LIN {X 0,Y 317.653,Z 381.301,A -85,B 0,C 180,E1 -15906.448,E2 -15906.448} C_VEL
LIN {X 0,Y 316.259,Z 393.2,A -85,B 0,C 180,E1 -15907.203,E2 -15907.203} C_VEL
LIN {X 0,Y 314.587,Z 404.894,A -85,B 0,C 180,E1 -15908.2,E2 -15908.2} C_VEL
LIN {X 0,Y 312.768,Z 416.27,A -85,B 0,C 180,E1 -15909.448,E2 -15909.448} C_VEL
LIN {X 0,Y 310.949,Z 426.626,A -85,B 0,C 180,E1 -15910.871,E2 -15910.871} C_VEL
LIN {X 0,Y 309.178,Z 435.992,A -85,B 0,C 180,E1 -15912.473,E2 -15912.473} C_VEL
LIN {X 0,Y 307.511,Z 445.132,A -85,B 0,C 180,E1 -15914.424,E2 -15914.424} C_VEL
LIN {X 0,Y 306.132,Z 452.545,A -85,B 0,C 180,E1 -15916.391,E2 -15916.391} C_VEL
LIN {X 0,Y 305.102,Z 457.603,A -85,B 0,C 180,E1 -15918.036,E2 -15918.036} C_VEL
LIN {X 0,Y 304.379,Z 462.545,A -85,B 0,C 180,E1 -15920.029,E2 -15920.029} C_VEL
LIN {X 0,Y 303.921,Z 466.357,A -85,B 0,C 180,E1 -15922.025,E2 -15922.025} C_VEL
LIN {X 0,Y 303.627,Z 469.641,A -85,B 0,C 180,E1 -15924.456,E2 -15924.456} C_VEL
LIN {X 0,Y 303.64,Z 470.96,A -85,B 0,C 180,E1 -15926.019,E2 -15926.019} C_VEL
LIN {X 0,Y 303.653,Z 471.66,A -85,B 0,C 180,E1 -15927.347,E2 -15927.347} C_VEL
LIN {X 0,Y 303.684,Z 471.954,A -85,B 0,C 180,E1 -15928.674,E2 -15928.674} C_VEL
LIN {X 0,Y 303.768,Z 471.795,A -85,B 0,C 180,E1 -15930,E2 -15930} C_VEL
LIN {X 0,Y 303.712,Z 471.218,A -85,B 0,C 180,E1 -15931.326,E2 -15931.326} C_VEL
LIN {X 0,Y 303.68,Z 470.233,A -85,B 0,C 180,E1 -15932.652,E2 -15932.652} C_VEL
LIN {X 0,Y 303.699,Z 468.813,A -85,B 0,C 180,E1 -15933.98,E2 -15933.98} C_VEL
LIN {X 0,Y 303.735,Z 466.181,A -85,B 0,C 180,E1 -15935.751,E2 -15935.751} C_VEL
LIN {X 0,Y 303.933,Z 461.681,A -85,B 0,C 180,E1 -15937.974,E2 -15937.974} C_VEL
LIN {X 0,Y 304.394,Z 455.299,A -85,B 0,C 180,E1 -15940.307,E2 -15940.307} C_VEL
LIN {X 0,Y 305.068,Z 448.32,A -85,B 0,C 180,E1 -15942.302,E2 -15942.302} C_VEL
LIN {X 0,Y 305.863,Z 441.179,A -85,B 0,C 180,E1 -15943.959,E2 -15943.959} C_VEL
LIN {X 0,Y 306.821,Z 433.215,A -85,B 0,C 180,E1 -15945.491,E2 -15945.491} C_VEL
LIN {X 0,Y 307.985,Z 423.186,A -85,B 0,C 180,E1 -15947.066,E2 -15947.066} C_VEL
LIN {X 0,Y 309.15,Z 412.766,A -85,B 0,C 180,E1 -15948.384,E2 -15948.384} C_VEL
LIN {X 0,Y 310.352,Z 401.577,A -85,B 0,C 180,E1 -15949.51,E2 -15949.51} C_VEL
LIN {X 0,Y 311.498,Z 389.171,A -85,B 0,C 180,E1 -15950.467,E2 -15950.467} C_VEL
LIN {X 0,Y 312.472,Z 375.35,A -85,B 0,C 180,E1 -15951.219,E2 -15951.219} C_VEL
LIN {X 0,Y 313.086,Z 362.94,A -85,B 0,C 180,E1 -15951.65,E2 -15951.65} C_VEL
LIN {X 0,Y 314.499,Z 301.548,A -85,B 0,C 180,E1 -15953.24,E2 -15953.24} C_VEL
LIN {X 0,Y 309.032,Z 259.907,A -85,B 0,C 180,E1 -15954.774,E2 -15954.774} C_VEL
LIN {X 0,Y 309.789,Z 252.83,A -85,B 0,C 180,E1 -15956.616,E2 -15956.616} C_VEL
LIN {X 0,Y 308.031,Z 243.339,A -85,B 0,C 180,E1 -15959.295,E2 -15959.295} C_VEL
LIN {X 0,Y 305.483,Z 231.433,A -85,B 0,C 180,E1 -15962.821,E2 -15962.821} C_VEL
LIN {X 0,Y 305.445,Z 231.435,A -85,B 0,C 180,E1 -15966.739,E2 -15966.739} C_VEL
LIN {X 0,Y 305.44,Z 231.436,A -85,B 0,C 180,E1 -15970.596,E2 -15970.596} C_VEL
LIN {X 0,Y 305.408,Z 231.444,A -85,B 0,C 180,E1 -15973.652,E2 -15973.652} C_VEL
LIN {X 0,Y 305.435,Z 231.439,A -85,B 0,C 180,E1 -15977.411,E2 -15977.411} C_VEL
LIN {X 0,Y 305.453,Z 231.438,A -85,B 0,C 180,E1 -15981.594,E2 -15981.594} C_VEL
LIN {X 0,Y 305.437,Z 231.436,A -85,B 0,C 180,E1 -15984.883,E2 -15984.883} C_VEL
LIN {X 0,Y 305.415,Z 231.439,A -85,B 0,C 180,E1 -15988.356,E2 -15988.356} C_VEL
LIN {X 0,Y 305.471,Z 231.434,A -85,B 0,C 180,E1 -15991.108,E2 -15991.108} C_VEL
LIN {X 0,Y 305.524,Z 231.424,A -85,B 0,C 180,E1 -15994.083,E2 -15994.083} C_VEL
LIN {X 0,Y 305.43,Z 231.437,A -85,B 0,C 180,E1 -15998.397,E2 -15998.397} C_VEL
LIN {X 0,Y 305.483,Z 231.434,A -85,B 0,C 180,E1 -16001.21,E2 -16001.21} C_VEL
LIN {X 0,Y 305.591,Z 231.419,A -85,B 0,C 180,E1 -16005.346,E2 -16005.346} C_VEL
LIN {X 0,Y 305.599,Z 231.418,A -85,B 0,C 180,E1 -16009.398,E2 -16009.398} C_VEL
LIN {X 0,Y 305.749,Z 231.397,A -85,B 0,C 180,E1 -16012.072,E2 -16012.072} C_VEL
LIN {X 0,Y 305.641,Z 231.412,A -85,B 0,C 180,E1 -16014.722,E2 -16014.722} C_VEL
LIN {X 0,Y 305.915,Z 231.376,A -85,B 0,C 180,E1 -16018.683,E2 -16018.683} C_VEL
LIN {X 0,Y 305.917,Z 231.376,A -85,B 0,C 180,E1 -16021.316,E2 -16021.316} C_VEL
LIN {X 0,Y 305.805,Z 231.393,A -85,B 0,C 180,E1 -16026.598,E2 -16026.598} C_VEL
LIN {X 0,Y 305.664,Z 231.408,A -85,B 0,C 180,E1 -16029.261,E2 -16029.261} C_VEL
LIN {X 0,Y 305.551,Z 231.421,A -85,B 0,C 180,E1 -16033.297,E2 -16033.297} C_VEL
LIN {X 0,Y 305.524,Z 231.423,A -85,B 0,C 180,E1 -16036.023,E2 -16036.023} C_VEL
LIN {X 0,Y 305.572,Z 231.414,A -85,B 0,C 180,E1 -16039.46,E2 -16039.46} C_VEL
LIN {X 0,Y 305.526,Z 231.424,A -85,B 0,C 180,E1 -16043.072,E2 -16043.072} C_VEL
LIN {X 0,Y 305.518,Z 231.428,A -85,B 0,C 180,E1 -16046.229,E2 -16046.229} C_VEL
LIN {X 0,Y 305.465,Z 231.433,A -85,B 0,C 180,E1 -16049.051,E2 -16049.051} C_VEL
LIN {X 0,Y 305.438,Z 231.435,A -85,B 0,C 180,E1 -16053.52,E2 -16053.52} C_VEL
LIN {X 0,Y 305.455,Z 231.431,A -85,B 0,C 180,E1 -16056.742,E2 -16056.742} C_VEL
LIN {X 0,Y 305.461,Z 231.43,A -85,B 0,C 180,E1 -16060.609,E2 -16060.609} C_VEL
LIN {X 0,Y 305.466,Z 231.432,A -85,B 0,C 180,E1 -16063.647,E2 -16063.647} C_VEL
LIN {X 0,Y 305.443,Z 231.435,A -85,B 0,C 180,E1 -16067.416,E2 -16067.416} C_VEL
LIN {X 0,Y 305.48,Z 231.432,A -85,B 0,C 180,E1 -16071.603,E2 -16071.603} C_VEL
LIN {X 0,Y 305.447,Z 231.433,A -85,B 0,C 180,E1 -16074.889,E2 -16074.889} C_VEL
LIN {X 0,Y 305.439,Z 231.434,A -85,B 0,C 180,E1 -16078.358,E2 -16078.358} C_VEL
LIN {X 0,Y 305.518,Z 231.425,A -85,B 0,C 180,E1 -16081.117,E2 -16081.117} C_VEL
LIN {X 0,Y 305.562,Z 231.422,A -85,B 0,C 180,E1 -16084.09,E2 -16084.09} C_VEL
LIN {X 0,Y 305.494,Z 231.428,A -85,B 0,C 180,E1 -16088.405,E2 -16088.405} C_VEL
LIN {X 0,Y 305.585,Z 231.418,A -85,B 0,C 180,E1 -16091.22,E2 -16091.22} C_VEL
LIN {X 0,Y 305.645,Z 231.414,A -85,B 0,C 180,E1 -16095.351,E2 -16095.351} C_VEL
LIN {X 0,Y 305.635,Z 231.415,A -85,B 0,C 180,E1 -16099.401,E2 -16099.401} C_VEL
LIN {X 0,Y 305.806,Z 231.39,A -85,B 0,C 180,E1 -16102.075,E2 -16102.075} C_VEL
LIN {X 0,Y 305.685,Z 231.406,A -85,B 0,C 180,E1 -16104.724,E2 -16104.724} C_VEL
LIN {X 0,Y 305.956,Z 231.372,A -85,B 0,C 180,E1 -16108.684,E2 -16108.684} C_VEL
LIN {X 0,Y 305.954,Z 231.375,A -85,B 0,C 180,E1 -16111.316,E2 -16111.316} C_VEL
LIN {X 0,Y 305.684,Z 231.409,A -85,B 0,C 180,E1 -16115.276,E2 -16115.276} C_VEL
LIN {X 0,Y 305.799,Z 231.391,A -85,B 0,C 180,E1 -16117.925,E2 -16117.925} C_VEL
LIN {X 0,Y 305.6,Z 231.416,A -85,B 0,C 180,E1 -16121.944,E2 -16121.944} C_VEL
LIN {X 0,Y 305.634,Z 231.416,A -85,B 0,C 180,E1 -16125.034,E2 -16125.034} C_VEL
LIN {X 0,Y 305.574,Z 231.423,A -85,B 0,C 180,E1 -16128.781,E2 -16128.781} C_VEL
LIN {X 0,Y 305.51,Z 231.43,A -85,B 0,C 180,E1 -16133.051,E2 -16133.051} C_VEL
LIN {X 0,Y 305.547,Z 231.505,A -85,B 0,C 180,E1 -16134.681,E2 -16134.681} C_VEL
LIN {X 0,Y 305.821,Z 232.846,A -85,B 0,C 180,E1 -16135.111,E2 -16135.111} C_VEL
LIN {X 0,Y 314.812,Z 258.671,A -85,B 0,C 180,E1 -16136.448,E2 -16136.448} C_VEL
LIN {X 0,Y 315.39,Z 262.897,A -85,B 0,C 180,E1 -16136.601,E2 -16136.601} C_VEL
LIN {X 0,Y 313.097,Z 340.52,A -85,B 0,C 180,E1 -16138.612,E2 -16138.612} C_VEL
LIN {X 0,Y 312.366,Z 354.527,A -85,B 0,C 180,E1 -16139.243,E2 -16139.243} C_VEL
LIN {X 0,Y 311.646,Z 367.397,A -85,B 0,C 180,E1 -16140.106,E2 -16140.106} C_VEL
LIN {X 0,Y 310.566,Z 379.68,A -85,B 0,C 180,E1 -16141.21,E2 -16141.21} C_VEL
LIN {X 0,Y 309.47,Z 390.887,A -85,B 0,C 180,E1 -16142.499,E2 -16142.499} C_VEL
LIN {X 0,Y 308.373,Z 400.89,A -85,B 0,C 180,E1 -16143.939,E2 -16143.939} C_VEL
LIN {X 0,Y 307.194,Z 410.679,A -85,B 0,C 180,E1 -16145.685,E2 -16145.685} C_VEL
LIN {X 0,Y 306.229,Z 418.724,A -85,B 0,C 180,E1 -16147.452,E2 -16147.452} C_VEL
LIN {X 0,Y 305.356,Z 425.655,A -85,B 0,C 180,E1 -16149.322,E2 -16149.322} C_VEL
LIN {X 0,Y 304.619,Z 432.271,A -85,B 0,C 180,E1 -16151.603,E2 -16151.603} C_VEL
LIN {X 0,Y 304.121,Z 437.291,A -85,B 0,C 180,E1 -16153.884,E2 -16153.884} C_VEL
LIN {X 0,Y 303.738,Z 440.726,A -85,B 0,C 180,E1 -16156.041,E2 -16156.041} C_VEL
LIN {X 0,Y 303.554,Z 442.645,A -85,B 0,C 180,E1 -16157.824,E2 -16157.824} C_VEL
LIN {X 0,Y 303.498,Z 443.917,A -85,B 0,C 180,E1 -16159.826,E2 -16159.826} C_VEL
LIN {X 0,Y 303.566,Z 444.255,A -85,B 0,C 180,E1 -16161.912,E2 -16161.912} C_VEL
LIN {X 0,Y 303.843,Z 443.556,A -85,B 0,C 180,E1 -16164.045,E2 -16164.045} C_VEL
LIN {X 0,Y 304.357,Z 441.614,A -85,B 0,C 180,E1 -16166.346,E2 -16166.346} C_VEL
LIN {X 0,Y 305.09,Z 438.685,A -85,B 0,C 180,E1 -16168.455,E2 -16168.455} C_VEL
LIN {X 0,Y 306.066,Z 434.158,A -85,B 0,C 180,E1 -16170.747,E2 -16170.747} C_VEL
LIN {X 0,Y 307.413,Z 427.954,A -85,B 0,C 180,E1 -16173.064,E2 -16173.064} C_VEL
LIN {X 0,Y 308.769,Z 421.574,A -85,B 0,C 180,E1 -16174.929,E2 -16174.929} C_VEL
LIN {X 0,Y 309.189,Z 419.694,A -85,B 0,C 180,E1 -16175.406,E2 -16175.406} C_VEL
LIN {X 0,Y 309.243,Z 416.212,A -85,B 0,C 180,E1 -16176.287,E2 -16176.287} C_VEL
LIN {X 0,Y 307.687,Z 410.378,A -85,B 0,C 180,E1 -16177.755,E2 -16177.755} C_VEL
LIN {X 0,Y 306.285,Z 404.047,A -85,B 0,C 180,E1 -16179.148,E2 -16179.148} C_VEL
LIN {X 0,Y 306.552,Z 399.726,A -85,B 0,C 180,E1 -16179.896,E2 -16179.896} C_VEL
LIN {X 0,Y 308.522,Z 388.726,A -85,B 0,C 180,E1 -16181.403,E2 -16181.403} C_VEL
LIN {X 0,Y 310.286,Z 376.54,A -85,B 0,C 180,E1 -16182.704,E2 -16182.704} C_VEL
LIN {X 0,Y 311.824,Z 363.991,A -85,B 0,C 180,E1 -16183.721,E2 -16183.721} C_VEL
LIN {X 0,Y 312.834,Z 351.349,A -85,B 0,C 180,E1 -16184.473,E2 -16184.473} C_VEL
LIN {X 0,Y 313.664,Z 337.768,A -85,B 0,C 180,E1 -16184.992,E2 -16184.992} C_VEL
LIN {X 0,Y 316.53,Z 269.283,A -85,B 0,C 180,E1 -16186.858,E2 -16186.858} C_VEL
LIN {X 0,Y 310.851,Z 256.38,A -85,B 0,C 180,E1 -16188.029,E2 -16188.029} C_VEL
LIN {X 0,Y 304.047,Z 243.48,A -85,B 0,C 180,E1 -16189.449,E2 -16189.449} C_VEL
LIN {X 0,Y 299.59,Z 235.645,A -85,B 0,C 180,E1 -16190.464,E2 -16190.464} C_VEL
LIN {X 0,Y 298.691,Z 232.281,A -85,B 0,C 180,E1 -16191.797,E2 -16191.797} C_VEL
LIN {X 0,Y 298.619,Z 232.287,A -85,B 0,C 180,E1 -16194.599,E2 -16194.599} C_VEL
LIN {X 0,Y 298.884,Z 232.253,A -85,B 0,C 180,E1 -16198.653,E2 -16198.653} C_VEL
LIN {X 0,Y 298.883,Z 232.253,A -85,B 0,C 180,E1 -16201.348,E2 -16201.348} C_VEL
LIN {X 0,Y 298.736,Z 232.272,A -85,B 0,C 180,E1 -16206.756,E2 -16206.756} C_VEL
LIN {X 0,Y 298.598,Z 232.29,A -85,B 0,C 180,E1 -16209.484,E2 -16209.484} C_VEL
LIN {X 0,Y 298.51,Z 232.298,A -85,B 0,C 180,E1 -16213.618,E2 -16213.618} C_VEL
LIN {X 0,Y 298.454,Z 232.306,A -85,B 0,C 180,E1 -16216.415,E2 -16216.415} C_VEL
LIN {X 0,Y 298.414,Z 232.311,A -85,B 0,C 180,E1 -16219.619,E2 -16219.619} C_VEL
LIN {X 0,Y 298.4,Z 232.307,A -85,B 0,C 180,E1 -16223.603,E2 -16223.603} C_VEL
LIN {X 0,Y 298.432,Z 232.305,A -85,B 0,C 180,E1 -16226.58,E2 -16226.58} C_VEL
LIN {X 0,Y 298.376,Z 232.31,A -85,B 0,C 180,E1 -16229.646,E2 -16229.646} C_VEL
LIN {X 0,Y 298.369,Z 232.314,A -85,B 0,C 180,E1 -16232.804,E2 -16232.804} C_VEL
LIN {X 0,Y 298.422,Z 232.313,A -85,B 0,C 180,E1 -16236.81,E2 -16236.81} C_VEL
LIN {X 0,Y 298.368,Z 232.316,A -85,B 0,C 180,E1 -16241.09,E2 -16241.09} C_VEL
LIN {X 0,Y 298.383,Z 232.312,A -85,B 0,C 180,E1 -16243.107,E2 -16243.107} C_VEL
LIN {X 0,Y 298.36,Z 232.319,A -85,B 0,C 180,E1 -16246.919,E2 -16246.919} C_VEL
LIN {X 0,Y 298.386,Z 232.317,A -85,B 0,C 180,E1 -16251.011,E2 -16251.011} C_VEL
LIN {X 0,Y 298.418,Z 232.317,A -85,B 0,C 180,E1 -16252.034,E2 -16252.034} C_VEL
LIN {X 0,Y 300.927,Z 240.915,A -85,B 0,C 180,E1 -16255.305,E2 -16255.305} C_VEL
LIN {X 0,Y 303.28,Z 250.22,A -85,B 0,C 180,E1 -16258.518,E2 -16258.518} C_VEL
LIN {X 0,Y 304.567,Z 256.176,A -85,B 0,C 180,E1 -16260.389,E2 -16260.389} C_VEL
LIN {X 0,Y 308.753,Z 265.73,A -85,B 0,C 180,E1 -16261.315,E2 -16261.315} C_VEL
LIN {X 0,Y 311.706,Z 280.086,A -85,B 0,C 180,E1 -16262.194,E2 -16262.194} C_VEL
LIN {X 0,Y 314.699,Z 299.499,A -85,B 0,C 180,E1 -16263.208,E2 -16263.208} C_VEL
LIN {X 0,Y 315.264,Z 306.524,A -85,B 0,C 180,E1 -16263.5,E2 -16263.5} C_VEL
LIN {X 0,Y 312.654,Z 367.047,A -85,B 0,C 180,E1 -16265.164,E2 -16265.164} C_VEL
LIN {X 0,Y 311.574,Z 380.568,A -85,B 0,C 180,E1 -16265.783,E2 -16265.783} C_VEL
LIN {X 0,Y 310.047,Z 392.522,A -85,B 0,C 180,E1 -16266.543,E2 -16266.543} C_VEL
LIN {X 0,Y 308.339,Z 404.235,A -85,B 0,C 180,E1 -16267.558,E2 -16267.558} C_VEL
LIN {X 0,Y 306.178,Z 416.902,A -85,B 0,C 180,E1 -16268.985,E2 -16268.985} C_VEL
LIN {X 0,Y 304.276,Z 427.056,A -85,B 0,C 180,E1 -16270.435,E2 -16270.435} C_VEL
LIN {X 0,Y 302.419,Z 436.278,A -85,B 0,C 180,E1 -16272.068,E2 -16272.068} C_VEL
LIN {X 0,Y 300.666,Z 445.323,A -85,B 0,C 180,E1 -16274.06,E2 -16274.06} C_VEL
LIN {X 0,Y 299.226,Z 452.637,A -85,B 0,C 180,E1 -16276.071,E2 -16276.071} C_VEL
LIN {X 0,Y 298.124,Z 457.607,A -85,B 0,C 180,E1 -16277.752,E2 -16277.752} C_VEL
LIN {X 0,Y 297.366,Z 462.462,A -85,B 0,C 180,E1 -16279.791,E2 -16279.791} C_VEL
LIN {X 0,Y 296.86,Z 466.206,A -85,B 0,C 180,E1 -16281.834,E2 -16281.834} C_VEL
LIN {X 0,Y 296.656,Z 468.148,A -85,B 0,C 180,E1 -16283.198,E2 -16283.198} C_VEL
LIN {X 0,Y 296.553,Z 469.623,A -85,B 0,C 180,E1 -16284.561,E2 -16284.561} C_VEL
LIN {X 0,Y 296.536,Z 470.696,A -85,B 0,C 180,E1 -16285.923,E2 -16285.923} C_VEL
LIN {X 0,Y 296.576,Z 471.37,A -85,B 0,C 180,E1 -16287.284,E2 -16287.284} C_VEL
LIN {X 0,Y 296.597,Z 471.61,A -85,B 0,C 180,E1 -16288.642,E2 -16288.642} C_VEL
LIN {X 0,Y 296.677,Z 471.415,A -85,B 0,C 180,E1 -16290,E2 -16290} C_VEL
LIN {X 0,Y 296.623,Z 470.809,A -85,B 0,C 180,E1 -16291.357,E2 -16291.357} C_VEL
LIN {X 0,Y 296.604,Z 469.793,A -85,B 0,C 180,E1 -16292.716,E2 -16292.716} C_VEL
LIN {X 0,Y 296.613,Z 468.308,A -85,B 0,C 180,E1 -16294.076,E2 -16294.076} C_VEL
LIN {X 0,Y 296.668,Z 465.877,A -85,B 0,C 180,E1 -16295.743,E2 -16295.743} C_VEL
LIN {X 0,Y 296.864,Z 461.036,A -85,B 0,C 180,E1 -16298.165,E2 -16298.165} C_VEL
LIN {X 0,Y 297.355,Z 454.573,A -85,B 0,C 180,E1 -16300.553,E2 -16300.553} C_VEL
LIN {X 0,Y 298.113,Z 447.504,A -85,B 0,C 180,E1 -16302.594,E2 -16302.594} C_VEL
LIN {X 0,Y 299.166,Z 438.604,A -85,B 0,C 180,E1 -16304.626,E2 -16304.626} C_VEL
LIN {X 0,Y 300.281,Z 429.289,A -85,B 0,C 180,E1 -16306.341,E2 -16306.341} C_VEL
LIN {X 0,Y 301.429,Z 419.421,A -85,B 0,C 180,E1 -16307.817,E2 -16307.817} C_VEL
LIN {X 0,Y 302.711,Z 408.296,A -85,B 0,C 180,E1 -16309.141,E2 -16309.141} C_VEL
LIN {X 0,Y 303.993,Z 395.922,A -85,B 0,C 180,E1 -16310.288,E2 -16310.288} C_VEL
LIN {X 0,Y 305.036,Z 384.322,A -85,B 0,C 180,E1 -16311.097,E2 -16311.097} C_VEL
LIN {X 0,Y 305.888,Z 371.068,A -85,B 0,C 180,E1 -16311.743,E2 -16311.743} C_VEL
LIN {X 0,Y 306.55,Z 351.56,A -85,B 0,C 180,E1 -16312.313,E2 -16312.313} C_VEL
LIN {X 0,Y 307.794,Z 302.784,A -85,B 0,C 180,E1 -16313.606,E2 -16313.606} C_VEL
LIN {X 0,Y 302.193,Z 259.713,A -85,B 0,C 180,E1 -16315.211,E2 -16315.211} C_VEL
LIN {X 0,Y 302.813,Z 254.711,A -85,B 0,C 180,E1 -16316.534,E2 -16316.534} C_VEL
LIN {X 0,Y 301.734,Z 247.77,A -85,B 0,C 180,E1 -16318.517,E2 -16318.517} C_VEL
LIN {X 0,Y 299.065,Z 235.374,A -85,B 0,C 180,E1 -16322.22,E2 -16322.22} C_VEL
LIN {X 0,Y 298.428,Z 232.311,A -85,B 0,C 180,E1 -16323.194,E2 -16323.194} C_VEL
LIN {X 0,Y 298.419,Z 232.311,A -85,B 0,C 180,E1 -16326.8,E2 -16326.8} C_VEL
LIN {X 0,Y 298.372,Z 232.316,A -85,B 0,C 180,E1 -16331.084,E2 -16331.084} C_VEL
LIN {X 0,Y 298.385,Z 232.315,A -85,B 0,C 180,E1 -16333.1,E2 -16333.1} C_VEL
LIN {X 0,Y 298.386,Z 232.315,A -85,B 0,C 180,E1 -16336.917,E2 -16336.917} C_VEL
LIN {X 0,Y 298.383,Z 232.315,A -85,B 0,C 180,E1 -16341.003,E2 -16341.003} C_VEL
LIN {X 0,Y 298.394,Z 232.315,A -85,B 0,C 180,E1 -16343.926,E2 -16343.926} C_VEL
LIN {X 0,Y 298.367,Z 232.318,A -85,B 0,C 180,E1 -16347.196,E2 -16347.196} C_VEL
LIN {X 0,Y 298.388,Z 232.314,A -85,B 0,C 180,E1 -16350.618,E2 -16350.618} C_VEL
LIN {X 0,Y 298.447,Z 232.309,A -85,B 0,C 180,E1 -16353.476,E2 -16353.476} C_VEL
LIN {X 0,Y 298.401,Z 232.312,A -85,B 0,C 180,E1 -16356.698,E2 -16356.698} C_VEL
LIN {X 0,Y 298.43,Z 232.309,A -85,B 0,C 180,E1 -16360.749,E2 -16360.749} C_VEL
LIN {X 0,Y 298.555,Z 232.293,A -85,B 0,C 180,E1 -16364.992,E2 -16364.992} C_VEL
LIN {X 0,Y 298.556,Z 232.298,A -85,B 0,C 180,E1 -16369.145,E2 -16369.145} C_VEL
LIN {X 0,Y 298.695,Z 232.276,A -85,B 0,C 180,E1 -16371.884,E2 -16371.884} C_VEL
LIN {X 0,Y 298.613,Z 232.287,A -85,B 0,C 180,E1 -16374.598,E2 -16374.598} C_VEL
LIN {X 0,Y 298.882,Z 232.251,A -85,B 0,C 180,E1 -16378.652,E2 -16378.652} C_VEL
LIN {X 0,Y 298.884,Z 232.251,A -85,B 0,C 180,E1 -16381.347,E2 -16381.347} C_VEL
LIN {X 0,Y 298.75,Z 232.273,A -85,B 0,C 180,E1 -16386.754,E2 -16386.754} C_VEL
LIN {X 0,Y 298.596,Z 232.288,A -85,B 0,C 180,E1 -16389.483,E2 -16389.483} C_VEL
LIN {X 0,Y 298.512,Z 232.296,A -85,B 0,C 180,E1 -16393.617,E2 -16393.617} C_VEL
LIN {X 0,Y 298.493,Z 232.3,A -85,B 0,C 180,E1 -16396.411,E2 -16396.411} C_VEL
LIN {X 0,Y 298.503,Z 232.293,A -85,B 0,C 180,E1 -16399.668,E2 -16399.668} C_VEL
LIN {X 0,Y 298.459,Z 232.303,A -85,B 0,C 180,E1 -16403.597,E2 -16403.597} C_VEL
LIN {X 0,Y 298.461,Z 232.308,A -85,B 0,C 180,E1 -16406.577,E2 -16406.577} C_VEL
LIN {X 0,Y 298.392,Z 232.314,A -85,B 0,C 180,E1 -16409.644,E2 -16409.644} C_VEL
LIN {X 0,Y 298.368,Z 232.316,A -85,B 0,C 180,E1 -16412.803,E2 -16412.803} C_VEL
LIN {X 0,Y 298.426,Z 232.306,A -85,B 0,C 180,E1 -16416.811,E2 -16416.811} C_VEL
LIN {X 0,Y 298.429,Z 232.304,A -85,B 0,C 180,E1 -16421.104,E2 -16421.104} C_VEL
LIN {X 0,Y 298.44,Z 232.304,A -85,B 0,C 180,E1 -16423.119,E2 -16423.119} C_VEL
LIN {X 0,Y 298.385,Z 232.314,A -85,B 0,C 180,E1 -16426.924,E2 -16426.924} C_VEL
LIN {X 0,Y 298.4,Z 232.312,A -85,B 0,C 180,E1 -16431.006,E2 -16431.006} C_VEL
LIN {X 0,Y 298.405,Z 232.314,A -85,B 0,C 180,E1 -16433.933,E2 -16433.933} C_VEL
LIN {X 0,Y 298.383,Z 232.315,A -85,B 0,C 180,E1 -16437.986,E2 -16437.986} C_VEL
LIN {X 0,Y 298.459,Z 232.308,A -85,B 0,C 180,E1 -16441.907,E2 -16441.907} C_VEL
LIN {X 0,Y 298.478,Z 232.303,A -85,B 0,C 180,E1 -16444.926,E2 -16444.926} C_VEL
LIN {X 0,Y 298.444,Z 232.309,A -85,B 0,C 180,E1 -16449.317,E2 -16449.317} C_VEL
LIN {X 0,Y 298.532,Z 232.295,A -85,B 0,C 180,E1 -16452.181,E2 -16452.181} C_VEL
LIN {X 0,Y 298.589,Z 232.29,A -85,B 0,C 180,E1 -16454.996,E2 -16454.996} C_VEL
LIN {X 0,Y 298.591,Z 232.291,A -85,B 0,C 180,E1 -16459.148,E2 -16459.148} C_VEL
LIN {X 0,Y 298.752,Z 232.269,A -85,B 0,C 180,E1 -16461.887,E2 -16461.887} C_VEL
LIN {X 0,Y 298.655,Z 232.281,A -85,B 0,C 180,E1 -16464.6,E2 -16464.6} C_VEL
LIN {X 0,Y 298.922,Z 232.248,A -85,B 0,C 180,E1 -16468.653,E2 -16468.653} C_VEL
LIN {X 0,Y 298.921,Z 232.251,A -85,B 0,C 180,E1 -16471.347,E2 -16471.347} C_VEL
LIN {X 0,Y 298.786,Z 232.267,A -85,B 0,C 180,E1 -16476.754,E2 -16476.754} C_VEL
LIN {X 0,Y 298.641,Z 232.284,A -85,B 0,C 180,E1 -16479.481,E2 -16479.481} C_VEL
LIN {X 0,Y 298.549,Z 232.295,A -85,B 0,C 180,E1 -16483.614,E2 -16483.614} C_VEL
LIN {X 0,Y 298.544,Z 232.296,A -85,B 0,C 180,E1 -16486.407,E2 -16486.407} C_VEL
LIN {X 0,Y 298.492,Z 232.301,A -85,B 0,C 180,E1 -16489.645,E2 -16489.645} C_VEL
LIN {X 0,Y 298.488,Z 232.432,A -85,B 0,C 180,E1 -16494.377,E2 -16494.377} C_VEL
LIN {X 0,Y 298.662,Z 233.26,A -85,B 0,C 180,E1 -16494.639,E2 -16494.639} C_VEL
LIN {X 0,Y 308.354,Z 261,A -85,B 0,C 180,E1 -16496.107,E2 -16496.107} C_VEL
LIN {X 0,Y 308.595,Z 264.999,A -85,B 0,C 180,E1 -16496.235,E2 -16496.235} C_VEL
LIN {X 0,Y 306.287,Z 341.206,A -85,B 0,C 180,E1 -16498.266,E2 -16498.266} C_VEL
LIN {X 0,Y 305.545,Z 354.566,A -85,B 0,C 180,E1 -16498.88,E2 -16498.88} C_VEL
LIN {X 0,Y 304.816,Z 367.133,A -85,B 0,C 180,E1 -16499.73,E2 -16499.73} C_VEL
LIN {X 0,Y 303.766,Z 379.095,A -85,B 0,C 180,E1 -16500.813,E2 -16500.813} C_VEL
LIN {X 0,Y 302.644,Z 390.441,A -85,B 0,C 180,E1 -16502.127,E2 -16502.127} C_VEL
LIN {X 0,Y 301.562,Z 400.073,A -85,B 0,C 180,E1 -16503.511,E2 -16503.511} C_VEL
LIN {X 0,Y 300.488,Z 408.891,A -85,B 0,C 180,E1 -16505.056,E2 -16505.056} C_VEL
LIN {X 0,Y 299.319,Z 417.995,A -85,B 0,C 180,E1 -16507.031,E2 -16507.031} C_VEL
LIN {X 0,Y 298.396,Z 425.28,A -85,B 0,C 180,E1 -16508.993,E2 -16508.993} C_VEL
LIN {X 0,Y 297.687,Z 431.076,A -85,B 0,C 180,E1 -16510.934,E2 -16510.934} C_VEL
LIN {X 0,Y 297.243,Z 435.658,A -85,B 0,C 180,E1 -16512.865,E2 -16512.865} C_VEL
LIN {X 0,Y 296.79,Z 439.936,A -85,B 0,C 180,E1 -16515.261,E2 -16515.261} C_VEL
LIN {X 0,Y 296.502,Z 442.437,A -85,B 0,C 180,E1 -16517.283,E2 -16517.283} C_VEL
LIN {X 0,Y 296.409,Z 444.006,A -85,B 0,C 180,E1 -16519.345,E2 -16519.345} C_VEL
LIN {X 0,Y 296.495,Z 444.605,A -85,B 0,C 180,E1 -16521.955,E2 -16521.955} C_VEL
LIN {X 0,Y 296.715,Z 444.208,A -85,B 0,C 180,E1 -16523.691,E2 -16523.691} C_VEL
LIN {X 0,Y 297.153,Z 442.738,A -85,B 0,C 180,E1 -16525.863,E2 -16525.863} C_VEL
LIN {X 0,Y 297.871,Z 440.032,A -85,B 0,C 180,E1 -16528.135,E2 -16528.135} C_VEL
LIN {X 0,Y 298.885,Z 435.961,A -85,B 0,C 180,E1 -16530.45,E2 -16530.45} C_VEL
LIN {X 0,Y 300.18,Z 430.284,A -85,B 0,C 180,E1 -16532.821,E2 -16532.821} C_VEL
LIN {X 0,Y 301.632,Z 423.988,A -85,B 0,C 180,E1 -16534.836,E2 -16534.836} C_VEL
LIN {X 0,Y 303.317,Z 416.235,A -85,B 0,C 180,E1 -16536.803,E2 -16536.803} C_VEL
LIN {X 0,Y 305.17,Z 406.751,A -85,B 0,C 180,E1 -16538.733,E2 -16538.733} C_VEL
LIN {X 0,Y 306.552,Z 399.726,A -85,B 0,C 180,E1 -16539.896,E2 -16539.896} C_VEL
LIN {X 0,Y 306.845,Z 395.246,A -85,B 0,C 180,E1 -16540.611,E2 -16540.611} C_VEL
LIN {X 0,Y 305.585,Z 387.875,A -85,B 0,C 180,E1 -16541.829,E2 -16541.829} C_VEL
LIN {X 0,Y 304.297,Z 380.11,A -85,B 0,C 180,E1 -16542.963,E2 -16542.963} C_VEL
LIN {X 0,Y 304.357,Z 375.029,A -85,B 0,C 180,E1 -16543.527,E2 -16543.527} C_VEL
LIN {X 0,Y 305.758,Z 363.86,A -85,B 0,C 180,E1 -16544.417,E2 -16544.417} C_VEL
LIN {X 0,Y 306.81,Z 351.06,A -85,B 0,C 180,E1 -16545.179,E2 -16545.179} C_VEL
LIN {X 0,Y 307.685,Z 337.548,A -85,B 0,C 180,E1 -16545.693,E2 -16545.693} C_VEL
LIN {X 0,Y 310.642,Z 271.349,A -85,B 0,C 180,E1 -16547.546,E2 -16547.546} C_VEL
LIN {X 0,Y 304.567,Z 257.828,A -85,B 0,C 180,E1 -16548.85,E2 -16548.85} C_VEL
LIN {X 0,Y 298.684,Z 246.862,A -85,B 0,C 180,E1 -16550.149,E2 -16550.149} C_VEL
LIN {X 0,Y 293.927,Z 238.832,A -85,B 0,C 180,E1 -16551.234,E2 -16551.234} C_VEL
LIN {X 0,Y 292.498,Z 236.175,A -85,B 0,C 180,E1 -16551.622,E2 -16551.622} C_VEL
LIN {X 0,Y 291.68,Z 233.153,A -85,B 0,C 180,E1 -16552.907,E2 -16552.907} C_VEL
LIN {X 0,Y 291.748,Z 233.143,A -85,B 0,C 180,E1 -16557.239,E2 -16557.239} C_VEL
LIN {X 0,Y 291.902,Z 233.126,A -85,B 0,C 180,E1 -16560,E2 -16560} C_VEL
LIN {X 0,Y 291.746,Z 233.143,A -85,B 0,C 180,E1 -16562.762,E2 -16562.762} C_VEL
LIN {X 0,Y 291.686,Z 233.151,A -85,B 0,C 180,E1 -16566.92,E2 -16566.92} C_VEL
LIN {X 0,Y 291.54,Z 233.17,A -85,B 0,C 180,E1 -16569.715,E2 -16569.715} C_VEL
LIN {X 0,Y 291.482,Z 233.171,A -85,B 0,C 180,E1 -16573.953,E2 -16573.953} C_VEL
LIN {X 0,Y 291.399,Z 233.182,A -85,B 0,C 180,E1 -16576.824,E2 -16576.824} C_VEL
LIN {X 0,Y 291.364,Z 233.187,A -85,B 0,C 180,E1 -16579.844,E2 -16579.844} C_VEL
LIN {X 0,Y 291.35,Z 233.187,A -85,B 0,C 180,E1 -16584.21,E2 -16584.21} C_VEL
LIN {X 0,Y 291.376,Z 233.185,A -85,B 0,C 180,E1 -16587.277,E2 -16587.277} C_VEL
LIN {X 0,Y 291.297,Z 233.195,A -85,B 0,C 180,E1 -16590.442,E2 -16590.442} C_VEL
LIN {X 0,Y 291.32,Z 233.196,A -85,B 0,C 180,E1 -16593.702,E2 -16593.702} C_VEL
LIN {X 0,Y 291.35,Z 233.193,A -85,B 0,C 180,E1 -16597.255,E2 -16597.255} C_VEL
LIN {X 0,Y 291.313,Z 233.193,A -85,B 0,C 180,E1 -16600.646,E2 -16600.646} C_VEL
LIN {X 0,Y 291.276,Z 233.203,A -85,B 0,C 180,E1 -16604.405,E2 -16604.405} C_VEL
LIN {X 0,Y 291.304,Z 233.198,A -85,B 0,C 180,E1 -16608.41,E2 -16608.41} C_VEL
LIN {X 0,Y 291.373,Z 233.368,A -85,B 0,C 180,E1 -16611.006,E2 -16611.006} C_VEL
LIN {X 0,Y 293.955,Z 241.697,A -85,B 0,C 180,E1 -16614.38,E2 -16614.38} C_VEL
LIN {X 0,Y 296.598,Z 252.27,A -85,B 0,C 180,E1 -16618.187,E2 -16618.187} C_VEL
LIN {X 0,Y 297.377,Z 255.701,A -85,B 0,C 180,E1 -16619.278,E2 -16619.278} C_VEL
LIN {X 0,Y 303.176,Z 268.304,A -85,B 0,C 180,E1 -16620.625,E2 -16620.625} C_VEL
LIN {X 0,Y 305.468,Z 279.057,A -85,B 0,C 180,E1 -16621.33,E2 -16621.33} C_VEL
LIN {X 0,Y 308.504,Z 298.418,A -85,B 0,C 180,E1 -16622.399,E2 -16622.399} C_VEL
LIN {X 0,Y 309.326,Z 306.983,A -85,B 0,C 180,E1 -16622.794,E2 -16622.794} C_VEL
LIN {X 0,Y 306.557,Z 367.325,A -85,B 0,C 180,E1 -16624.499,E2 -16624.499} C_VEL
LIN {X 0,Y 305.322,Z 381.362,A -85,B 0,C 180,E1 -16625.163,E2 -16625.163} C_VEL
LIN {X 0,Y 303.765,Z 392.964,A -85,B 0,C 180,E1 -16625.937,E2 -16625.937} C_VEL
LIN {X 0,Y 301.849,Z 405.276,A -85,B 0,C 180,E1 -16627.048,E2 -16627.048} C_VEL
LIN {X 0,Y 299.866,Z 416.414,A -85,B 0,C 180,E1 -16628.34,E2 -16628.34} C_VEL
LIN {X 0,Y 297.782,Z 426.564,A -85,B 0,C 180,E1 -16629.81,E2 -16629.81} C_VEL
LIN {X 0,Y 295.682,Z 436.596,A -85,B 0,C 180,E1 -16631.645,E2 -16631.645} C_VEL
LIN {X 0,Y 293.823,Z 445.514,A -85,B 0,C 180,E1 -16633.679,E2 -16633.679} C_VEL
LIN {X 0,Y 292.326,Z 452.7,A -85,B 0,C 180,E1 -16635.735,E2 -16635.735} C_VEL
LIN {X 0,Y 291.158,Z 457.632,A -85,B 0,C 180,E1 -16637.454,E2 -16637.454} C_VEL
LIN {X 0,Y 290.367,Z 462.41,A -85,B 0,C 180,E1 -16639.542,E2 -16639.542} C_VEL
LIN {X 0,Y 289.82,Z 466.082,A -85,B 0,C 180,E1 -16641.635,E2 -16641.635} C_VEL
LIN {X 0,Y 289.581,Z 467.951,A -85,B 0,C 180,E1 -16643.031,E2 -16643.031} C_VEL
LIN {X 0,Y 289.477,Z 469.468,A -85,B 0,C 180,E1 -16644.513,E2 -16644.513} C_VEL
LIN {X 0,Y 289.498,Z 471.075,A -85,B 0,C 180,E1 -16647.217,E2 -16647.217} C_VEL
LIN {X 0,Y 289.512,Z 471.26,A -85,B 0,C 180,E1 -16648.609,E2 -16648.609} C_VEL
LIN {X 0,Y 289.587,Z 471.036,A -85,B 0,C 180,E1 -16650,E2 -16650} C_VEL
LIN {X 0,Y 289.538,Z 470.4,A -85,B 0,C 180,E1 -16651.391,E2 -16651.391} C_VEL
LIN {X 0,Y 289.528,Z 469.342,A -85,B 0,C 180,E1 -16652.782,E2 -16652.782} C_VEL
LIN {X 0,Y 289.531,Z 467.803,A -85,B 0,C 180,E1 -16654.175,E2 -16654.175} C_VEL
LIN {X 0,Y 289.62,Z 464.659,A -85,B 0,C 180,E1 -16656.268,E2 -16656.268} C_VEL
LIN {X 0,Y 289.817,Z 460.385,A -85,B 0,C 180,E1 -16658.365,E2 -16658.365} C_VEL
LIN {X 0,Y 290.321,Z 453.835,A -85,B 0,C 180,E1 -16660.812,E2 -16660.812} C_VEL
LIN {X 0,Y 291.163,Z 446.64,A -85,B 0,C 180,E1 -16662.9,E2 -16662.9} C_VEL
LIN {X 0,Y 292.276,Z 437.614,A -85,B 0,C 180,E1 -16664.979,E2 -16664.979} C_VEL
LIN {X 0,Y 293.297,Z 429.133,A -85,B 0,C 180,E1 -16666.566,E2 -16666.566} C_VEL
LIN {X 0,Y 294.462,Z 419.323,A -85,B 0,C 180,E1 -16668.074,E2 -16668.074} C_VEL
LIN {X 0,Y 295.777,Z 408.263,A -85,B 0,C 180,E1 -16669.428,E2 -16669.428} C_VEL
LIN {X 0,Y 297.104,Z 395.965,A -85,B 0,C 180,E1 -16670.599,E2 -16670.599} C_VEL
LIN {X 0,Y 298.246,Z 383.099,A -85,B 0,C 180,E1 -16671.511,E2 -16671.511} C_VEL
LIN {X 0,Y 299.182,Z 369.453,A -85,B 0,C 180,E1 -16672.165,E2 -16672.165} C_VEL
LIN {X 0,Y 300.315,Z 332.242,A -85,B 0,C 180,E1 -16673.212,E2 -16673.212} C_VEL
LIN {X 0,Y 300.978,Z 303.014,A -85,B 0,C 180,E1 -16674.014,E2 -16674.014} C_VEL
LIN {X 0,Y 295.373,Z 259.388,A -85,B 0,C 180,E1 -16675.695,E2 -16675.695} C_VEL
LIN {X 0,Y 295.82,Z 255.233,A -85,B 0,C 180,E1 -16676.83,E2 -16676.83} C_VEL
LIN {X 0,Y 294.278,Z 246.833,A -85,B 0,C 180,E1 -16679.31,E2 -16679.31} C_VEL
LIN {X 0,Y 291.491,Z 233.685,A -85,B 0,C 180,E1 -16683.371,E2 -16683.371} C_VEL
LIN {X 0,Y 291.406,Z 233.187,A -85,B 0,C 180,E1 -16683.534,E2 -16683.534} C_VEL
LIN {X 0,Y 291.351,Z 233.192,A -85,B 0,C 180,E1 -16687.247,E2 -16687.247} C_VEL
LIN {X 0,Y 291.318,Z 233.195,A -85,B 0,C 180,E1 -16690.639,E2 -16690.639} C_VEL
LIN {X 0,Y 291.275,Z 233.202,A -85,B 0,C 180,E1 -16694.398,E2 -16694.398} C_VEL
LIN {X 0,Y 291.307,Z 233.197,A -85,B 0,C 180,E1 -16698.401,E2 -16698.401} C_VEL
LIN {X 0,Y 291.332,Z 233.194,A -85,B 0,C 180,E1 -16701.154,E2 -16701.154} C_VEL
LIN {X 0,Y 291.339,Z 233.191,A -85,B 0,C 180,E1 -16704.622,E2 -16704.622} C_VEL
LIN {X 0,Y 291.34,Z 233.194,A -85,B 0,C 180,E1 -16707.946,E2 -16707.946} C_VEL
LIN {X 0,Y 291.335,Z 233.195,A -85,B 0,C 180,E1 -16711.153,E2 -16711.153} C_VEL
LIN {X 0,Y 291.378,Z 233.185,A -85,B 0,C 180,E1 -16714.268,E2 -16714.268} C_VEL
LIN {X 0,Y 291.339,Z 233.196,A -85,B 0,C 180,E1 -16717.296,E2 -16717.296} C_VEL
LIN {X 0,Y 291.359,Z 233.189,A -85,B 0,C 180,E1 -16720.263,E2 -16720.263} C_VEL
LIN {X 0,Y 291.467,Z 233.172,A -85,B 0,C 180,E1 -16724.664,E2 -16724.664} C_VEL
LIN {X 0,Y 291.5,Z 233.174,A -85,B 0,C 180,E1 -16728.879,E2 -16728.879} C_VEL
LIN {X 0,Y 291.644,Z 233.155,A -85,B 0,C 180,E1 -16731.686,E2 -16731.686} C_VEL
LIN {X 0,Y 291.584,Z 233.161,A -85,B 0,C 180,E1 -16734.467,E2 -16734.467} C_VEL
LIN {X 0,Y 291.849,Z 233.125,A -85,B 0,C 180,E1 -16738.62,E2 -16738.62} C_VEL
LIN {X 0,Y 291.851,Z 233.126,A -85,B 0,C 180,E1 -16741.379,E2 -16741.379} C_VEL
LIN {X 0,Y 291.697,Z 233.151,A -85,B 0,C 180,E1 -16746.919,E2 -16746.919} C_VEL
LIN {X 0,Y 291.538,Z 233.167,A -85,B 0,C 180,E1 -16749.714,E2 -16749.714} C_VEL
LIN {X 0,Y 291.483,Z 233.172,A -85,B 0,C 180,E1 -16753.952,E2 -16753.952} C_VEL
LIN {X 0,Y 291.446,Z 233.173,A -85,B 0,C 180,E1 -16758.269,E2 -16758.269} C_VEL
LIN {X 0,Y 291.387,Z 233.181,A -85,B 0,C 180,E1 -16761.209,E2 -16761.209} C_VEL
LIN {X 0,Y 291.408,Z 233.183,A -85,B 0,C 180,E1 -16764.204,E2 -16764.204} C_VEL
LIN {X 0,Y 291.394,Z 233.185,A -85,B 0,C 180,E1 -16767.274,E2 -16767.274} C_VEL
LIN {X 0,Y 291.309,Z 233.2,A -85,B 0,C 180,E1 -16770.44,E2 -16770.44} C_VEL
LIN {X 0,Y 291.318,Z 233.194,A -85,B 0,C 180,E1 -16773.701,E2 -16773.701} C_VEL
LIN {X 0,Y 291.363,Z 233.184,A -85,B 0,C 180,E1 -16777.259,E2 -16777.259} C_VEL
LIN {X 0,Y 291.378,Z 233.182,A -85,B 0,C 180,E1 -16780.634,E2 -16780.634} C_VEL
LIN {X 0,Y 291.314,Z 233.196,A -85,B 0,C 180,E1 -16784.397,E2 -16784.397} C_VEL
LIN {X 0,Y 291.315,Z 233.197,A -85,B 0,C 180,E1 -16788.406,E2 -16788.406} C_VEL
LIN {X 0,Y 291.349,Z 233.191,A -85,B 0,C 180,E1 -16791.163,E2 -16791.163} C_VEL
LIN {X 0,Y 291.348,Z 233.188,A -85,B 0,C 180,E1 -16794.629,E2 -16794.629} C_VEL
LIN {X 0,Y 291.36,Z 233.189,A -85,B 0,C 180,E1 -16797.953,E2 -16797.953} C_VEL
LIN {X 0,Y 291.376,Z 233.186,A -85,B 0,C 180,E1 -16801.161,E2 -16801.161} C_VEL
LIN {X 0,Y 291.409,Z 233.184,A -85,B 0,C 180,E1 -16804.274,E2 -16804.274} C_VEL
LIN {X 0,Y 291.375,Z 233.19,A -85,B 0,C 180,E1 -16807.302,E2 -16807.302} C_VEL
LIN {X 0,Y 291.452,Z 233.175,A -85,B 0,C 180,E1 -16810.272,E2 -16810.272} C_VEL
LIN {X 0,Y 291.551,Z 233.165,A -85,B 0,C 180,E1 -16814.625,E2 -16814.625} C_VEL
LIN {X 0,Y 291.534,Z 233.168,A -85,B 0,C 180,E1 -16818.882,E2 -16818.882} C_VEL
LIN {X 0,Y 291.704,Z 233.149,A -85,B 0,C 180,E1 -16821.689,E2 -16821.689} C_VEL
LIN {X 0,Y 291.626,Z 233.157,A -85,B 0,C 180,E1 -16824.469,E2 -16824.469} C_VEL
LIN {X 0,Y 291.888,Z 233.124,A -85,B 0,C 180,E1 -16828.621,E2 -16828.621} C_VEL
LIN {X 0,Y 291.887,Z 233.126,A -85,B 0,C 180,E1 -16831.38,E2 -16831.38} C_VEL
LIN {X 0,Y 291.735,Z 233.146,A -85,B 0,C 180,E1 -16836.918,E2 -16836.918} C_VEL
LIN {X 0,Y 291.577,Z 233.163,A -85,B 0,C 180,E1 -16839.713,E2 -16839.713} C_VEL
LIN {X 0,Y 291.519,Z 233.171,A -85,B 0,C 180,E1 -16843.949,E2 -16843.949} C_VEL
LIN {X 0,Y 291.482,Z 233.179,A -85,B 0,C 180,E1 -16846.816,E2 -16846.816} C_VEL
LIN {X 0,Y 291.445,Z 233.179,A -85,B 0,C 180,E1 -16849.873,E2 -16849.873} C_VEL
LIN {X 0,Y 291.456,Z 233.28,A -85,B 0,C 180,E1 -16854.04,E2 -16854.04} C_VEL
LIN {X 0,Y 291.614,Z 234.1,A -85,B 0,C 180,E1 -16854.157,E2 -16854.157} C_VEL
LIN {X 0,Y 299.848,Z 257.183,A -85,B 0,C 180,E1 -16855.433,E2 -16855.433} C_VEL
LIN {X 0,Y 301.894,Z 263.368,A -85,B 0,C 180,E1 -16855.752,E2 -16855.752} C_VEL
LIN {X 0,Y 299.477,Z 341.91,A -85,B 0,C 180,E1 -16857.904,E2 -16857.904} C_VEL
LIN {X 0,Y 298.715,Z 355.355,A -85,B 0,C 180,E1 -16858.545,E2 -16858.545} C_VEL
LIN {X 0,Y 297.913,Z 368.084,A -85,B 0,C 180,E1 -16859.439,E2 -16859.439} C_VEL
LIN {X 0,Y 296.783,Z 380.447,A -85,B 0,C 180,E1 -16860.602,E2 -16860.602} C_VEL
LIN {X 0,Y 295.641,Z 391.477,A -85,B 0,C 180,E1 -16861.929,E2 -16861.929} C_VEL
LIN {X 0,Y 294.463,Z 401.725,A -85,B 0,C 180,E1 -16863.474,E2 -16863.474} C_VEL
LIN {X 0,Y 293.11,Z 411.938,A -85,B 0,C 180,E1 -16865.391,E2 -16865.391} C_VEL
LIN {X 0,Y 291.981,Z 420.533,A -85,B 0,C 180,E1 -16867.411,E2 -16867.411} C_VEL
LIN {X 0,Y 291.142,Z 427.383,A -85,B 0,C 180,E1 -16869.425,E2 -16869.425} C_VEL
LIN {X 0,Y 290.466,Z 432.802,A -85,B 0,C 180,E1 -16871.405,E2 -16871.405} C_VEL
LIN {X 0,Y 290.042,Z 437.068,A -85,B 0,C 180,E1 -16873.371,E2 -16873.371} C_VEL
LIN {X 0,Y 289.682,Z 440.285,A -85,B 0,C 180,E1 -16875.286,E2 -16875.286} C_VEL
LIN {X 0,Y 289.431,Z 442.591,A -85,B 0,C 180,E1 -16877.165,E2 -16877.165} C_VEL
LIN {X 0,Y 289.339,Z 444.07,A -85,B 0,C 180,E1 -16879.018,E2 -16879.018} C_VEL
LIN {X 0,Y 289.331,Z 444.867,A -85,B 0,C 180,E1 -16881.006,E2 -16881.006} C_VEL
LIN {X 0,Y 289.538,Z 444.776,A -85,B 0,C 180,E1 -16883.219,E2 -16883.219} C_VEL
LIN {X 0,Y 289.956,Z 443.609,A -85,B 0,C 180,E1 -16885.488,E2 -16885.488} C_VEL
LIN {X 0,Y 290.681,Z 441.195,A -85,B 0,C 180,E1 -16887.866,E2 -16887.866} C_VEL
LIN {X 0,Y 291.657,Z 437.641,A -85,B 0,C 180,E1 -16890.157,E2 -16890.157} C_VEL
LIN {X 0,Y 292.949,Z 432.441,A -85,B 0,C 180,E1 -16892.567,E2 -16892.567} C_VEL
LIN {X 0,Y 294.671,Z 425.441,A -85,B 0,C 180,E1 -16894.987,E2 -16894.987} C_VEL
LIN {X 0,Y 296.321,Z 418.542,A -85,B 0,C 180,E1 -16896.87,E2 -16896.87} C_VEL
LIN {X 0,Y 297.939,Z 411.011,A -85,B 0,C 180,E1 -16898.555,E2 -16898.555} C_VEL
LIN {X 0,Y 299.863,Z 401.664,A -85,B 0,C 180,E1 -16900.246,E2 -16900.246} C_VEL
LIN {X 0,Y 302.032,Z 390.336,A -85,B 0,C 180,E1 -16901.866,E2 -16901.866} C_VEL
LIN {X 0,Y 303.869,Z 378.513,A -85,B 0,C 180,E1 -16903.196,E2 -16903.196} C_VEL
LIN {X 0,Y 304.357,Z 375.029,A -85,B 0,C 180,E1 -16903.527,E2 -16903.527} C_VEL
LIN {X 0,Y 304.479,Z 369.827,A -85,B 0,C 180,E1 -16904.056,E2 -16904.056} C_VEL
LIN {X 0,Y 303.047,Z 361.313,A -85,B 0,C 180,E1 -16904.976,E2 -16904.976} C_VEL
LIN {X 0,Y 301.422,Z 352.526,A -85,B 0,C 180,E1 -16905.775,E2 -16905.775} C_VEL
LIN {X 0,Y 301.215,Z 346.903,A -85,B 0,C 180,E1 -16906.105,E2 -16906.105} C_VEL
LIN {X 0,Y 302.206,Z 327.234,A -85,B 0,C 180,E1 -16906.733,E2 -16906.733} C_VEL
LIN {X 0,Y 304.759,Z 273.487,A -85,B 0,C 180,E1 -16908.265,E2 -16908.265} C_VEL
LIN {X 0,Y 299.279,Z 261.202,A -85,B 0,C 180,E1 -16909.518,E2 -16909.518} C_VEL
LIN {X 0,Y 292.685,Z 248.904,A -85,B 0,C 180,E1 -16911.043,E2 -16911.043} C_VEL
LIN {X 0,Y 287.46,Z 240.293,A -85,B 0,C 180,E1 -16912.317,E2 -16912.317} C_VEL
LIN {X 0,Y 285.445,Z 236.704,A -85,B 0,C 180,E1 -16912.885,E2 -16912.885} C_VEL
LIN {X 0,Y 284.563,Z 234.041,A -85,B 0,C 180,E1 -16914.153,E2 -16914.153} C_VEL
LIN {X 0,Y 284.817,Z 234.006,A -85,B 0,C 180,E1 -16918.587,E2 -16918.587} C_VEL
LIN {X 0,Y 284.817,Z 234.006,A -85,B 0,C 180,E1 -16921.414,E2 -16921.414} C_VEL
LIN {X 0,Y 284.639,Z 234.031,A -85,B 0,C 180,E1 -16927.092,E2 -16927.092} C_VEL
LIN {X 0,Y 284.486,Z 234.048,A -85,B 0,C 180,E1 -16929.959,E2 -16929.959} C_VEL
LIN {X 0,Y 284.431,Z 234.048,A -85,B 0,C 180,E1 -16934.306,E2 -16934.306} C_VEL
LIN {X 0,Y 284.303,Z 234.072,A -85,B 0,C 180,E1 -16938.746,E2 -16938.746} C_VEL
LIN {X 0,Y 284.304,Z 234.063,A -85,B 0,C 180,E1 -16943.299,E2 -16943.299} C_VEL
LIN {X 0,Y 284.354,Z 234.059,A -85,B 0,C 180,E1 -16947.168,E2 -16947.168} C_VEL
LIN {X 0,Y 284.262,Z 234.075,A -85,B 0,C 180,E1 -16951.279,E2 -16951.279} C_VEL
LIN {X 0,Y 284.32,Z 234.062,A -85,B 0,C 180,E1 -16955.351,E2 -16955.351} C_VEL
LIN {X 0,Y 284.287,Z 234.069,A -85,B 0,C 180,E1 -16958.173,E2 -16958.173} C_VEL
LIN {X 0,Y 284.252,Z 234.078,A -85,B 0,C 180,E1 -16962.127,E2 -16962.127} C_VEL
LIN {X 0,Y 284.242,Z 234.077,A -85,B 0,C 180,E1 -16966.193,E2 -16966.193} C_VEL
LIN {X 0,Y 284.314,Z 234.237,A -85,B 0,C 180,E1 -16969.804,E2 -16969.804} C_VEL
LIN {X 0,Y 286.825,Z 242.407,A -85,B 0,C 180,E1 -16973.316,E2 -16973.316} C_VEL
LIN {X 0,Y 288.679,Z 249.171,A -85,B 0,C 180,E1 -16975.952,E2 -16975.952} C_VEL
LIN {X 0,Y 290.139,Z 255.099,A -85,B 0,C 180,E1 -16978.06,E2 -16978.06} C_VEL
LIN {X 0,Y 296.75,Z 268.834,A -85,B 0,C 180,E1 -16979.676,E2 -16979.676} C_VEL
LIN {X 0,Y 298.37,Z 273.273,A -85,B 0,C 180,E1 -16980.092,E2 -16980.092} C_VEL
LIN {X 0,Y 301.666,Z 292.343,A -85,B 0,C 180,E1 -16981.272,E2 -16981.272} C_VEL
LIN {X 0,Y 303.464,Z 306.704,A -85,B 0,C 180,E1 -16982.018,E2 -16982.018} C_VEL
LIN {X 0,Y 300.674,Z 365.897,A -85,B 0,C 180,E1 -16983.73,E2 -16983.73} C_VEL
LIN {X 0,Y 299.415,Z 380.13,A -85,B 0,C 180,E1 -16984.406,E2 -16984.406} C_VEL
LIN {X 0,Y 297.654,Z 392.447,A -85,B 0,C 180,E1 -16985.225,E2 -16985.225} C_VEL
LIN {X 0,Y 295.669,Z 404.757,A -85,B 0,C 180,E1 -16986.355,E2 -16986.355} C_VEL
LIN {X 0,Y 293.579,Z 415.929,A -85,B 0,C 180,E1 -16987.667,E2 -16987.667} C_VEL
LIN {X 0,Y 291.389,Z 426.112,A -85,B 0,C 180,E1 -16989.163,E2 -16989.163} C_VEL
LIN {X 0,Y 289.337,Z 435.342,A -85,B 0,C 180,E1 -16990.86,E2 -16990.86} C_VEL
LIN {X 0,Y 287.294,Z 444.396,A -85,B 0,C 180,E1 -16992.931,E2 -16992.931} C_VEL
LIN {X 0,Y 285.671,Z 451.734,A -85,B 0,C 180,E1 -16995.031,E2 -16995.031} C_VEL
LIN {X 0,Y 284.205,Z 457.634,A -85,B 0,C 180,E1 -16997.142,E2 -16997.142} C_VEL
LIN {X 0,Y 283.353,Z 462.335,A -85,B 0,C 180,E1 -16999.28,E2 -16999.28} C_VEL
LIN {X 0,Y 282.77,Z 465.945,A -85,B 0,C 180,E1 -17001.425,E2 -17001.425} C_VEL
LIN {X 0,Y 282.386,Z 469.172,A -85,B 0,C 180,E1 -17004.287,E2 -17004.287} C_VEL
LIN {X 0,Y 282.344,Z 470.182,A -85,B 0,C 180,E1 -17005.718,E2 -17005.718} C_VEL
LIN {X 0,Y 282.422,Z 470.764,A -85,B 0,C 180,E1 -17007.147,E2 -17007.147} C_VEL
LIN {X 0,Y 282.43,Z 470.909,A -85,B 0,C 180,E1 -17008.574,E2 -17008.574} C_VEL
LIN {X 0,Y 282.5,Z 470.654,A -85,B 0,C 180,E1 -17010,E2 -17010} C_VEL
LIN {X 0,Y 282.455,Z 469.988,A -85,B 0,C 180,E1 -17011.425,E2 -17011.425} C_VEL
LIN {X 0,Y 282.455,Z 468.871,A -85,B 0,C 180,E1 -17012.852,E2 -17012.852} C_VEL
LIN {X 0,Y 282.434,Z 466.34,A -85,B 0,C 180,E1 -17015.011,E2 -17015.011} C_VEL
LIN {X 0,Y 282.583,Z 462.783,A -85,B 0,C 180,E1 -17017.142,E2 -17017.142} C_VEL
LIN {X 0,Y 282.866,Z 458.025,A -85,B 0,C 180,E1 -17019.293,E2 -17019.293} C_VEL
LIN {X 0,Y 283.365,Z 451.95,A -85,B 0,C 180,E1 -17021.443,E2 -17021.443} C_VEL
LIN {X 0,Y 284.361,Z 444.372,A -85,B 0,C 180,E1 -17023.578,E2 -17023.578} C_VEL
LIN {X 0,Y 285.393,Z 436.622,A -85,B 0,C 180,E1 -17025.349,E2 -17025.349} C_VEL
LIN {X 0,Y 286.294,Z 429.068,A -85,B 0,C 180,E1 -17026.786,E2 -17026.786} C_VEL
LIN {X 0,Y 287.497,Z 419.219,A -85,B 0,C 180,E1 -17028.343,E2 -17028.343} C_VEL
LIN {X 0,Y 288.857,Z 408.232,A -85,B 0,C 180,E1 -17029.727,E2 -17029.727} C_VEL
LIN {X 0,Y 290.223,Z 396.008,A -85,B 0,C 180,E1 -17030.925,E2 -17030.925} C_VEL
LIN {X 0,Y 291.389,Z 383.318,A -85,B 0,C 180,E1 -17031.857,E2 -17031.857} C_VEL
LIN {X 0,Y 292.321,Z 369.925,A -85,B 0,C 180,E1 -17032.527,E2 -17032.527} C_VEL
LIN {X 0,Y 293.058,Z 347.153,A -85,B 0,C 180,E1 -17033.213,E2 -17033.213} C_VEL
LIN {X 0,Y 294.262,Z 304.009,A -85,B 0,C 180,E1 -17034.417,E2 -17034.417} C_VEL
LIN {X 0,Y 288.587,Z 259,A -85,B 0,C 180,E1 -17036.214,E2 -17036.214} C_VEL
LIN {X 0,Y 288.746,Z 255.692,A -85,B 0,C 180,E1 -17037.149,E2 -17037.149} C_VEL
LIN {X 0,Y 286.859,Z 245.86,A -85,B 0,C 180,E1 -17040.145,E2 -17040.145} C_VEL
LIN {X 0,Y 284.353,Z 234.066,A -85,B 0,C 180,E1 -17043.942,E2 -17043.942} C_VEL
LIN {X 0,Y 284.293,Z 234.073,A -85,B 0,C 180,E1 -17048.167,E2 -17048.167} C_VEL
LIN {X 0,Y 284.255,Z 234.078,A -85,B 0,C 180,E1 -17052.12,E2 -17052.12} C_VEL
LIN {X 0,Y 284.24,Z 234.079,A -85,B 0,C 180,E1 -17056.186,E2 -17056.186} C_VEL
LIN {X 0,Y 284.289,Z 234.073,A -85,B 0,C 180,E1 -17060.02,E2 -17060.02} C_VEL
LIN {X 0,Y 284.31,Z 234.072,A -85,B 0,C 180,E1 -17063.61,E2 -17063.61} C_VEL
LIN {X 0,Y 284.264,Z 234.074,A -85,B 0,C 180,E1 -17067.193,E2 -17067.193} C_VEL
LIN {X 0,Y 284.319,Z 234.067,A -85,B 0,C 180,E1 -17070.371,E2 -17070.371} C_VEL
LIN {X 0,Y 284.335,Z 234.066,A -85,B 0,C 180,E1 -17073.582,E2 -17073.582} C_VEL
LIN {X 0,Y 284.303,Z 234.068,A -85,B 0,C 180,E1 -17076.701,E2 -17076.701} C_VEL
LIN {X 0,Y 284.299,Z 234.072,A -85,B 0,C 180,E1 -17081.254,E2 -17081.254} C_VEL
LIN {X 0,Y 284.43,Z 234.051,A -85,B 0,C 180,E1 -17085.694,E2 -17085.694} C_VEL
LIN {X 0,Y 284.485,Z 234.046,A -85,B 0,C 180,E1 -17090.041,E2 -17090.041} C_VEL
LIN {X 0,Y 284.644,Z 234.029,A -85,B 0,C 180,E1 -17092.908,E2 -17092.908} C_VEL
LIN {X 0,Y 284.815,Z 234,A -85,B 0,C 180,E1 -17098.586,E2 -17098.586} C_VEL
LIN {X 0,Y 284.817,Z 234.001,A -85,B 0,C 180,E1 -17101.413,E2 -17101.413} C_VEL
LIN {X 0,Y 284.648,Z 234.028,A -85,B 0,C 180,E1 -17107.091,E2 -17107.091} C_VEL
LIN {X 0,Y 284.484,Z 234.046,A -85,B 0,C 180,E1 -17109.958,E2 -17109.958} C_VEL
LIN {X 0,Y 284.436,Z 234.051,A -85,B 0,C 180,E1 -17114.305,E2 -17114.305} C_VEL
LIN {X 0,Y 284.39,Z 234.051,A -85,B 0,C 180,E1 -17118.739,E2 -17118.739} C_VEL
LIN {X 0,Y 284.341,Z 234.058,A -85,B 0,C 180,E1 -17121.761,E2 -17121.761} C_VEL
LIN {X 0,Y 284.338,Z 234.064,A -85,B 0,C 180,E1 -17124.846,E2 -17124.846} C_VEL
LIN {X 0,Y 284.303,Z 234.07,A -85,B 0,C 180,E1 -17128.013,E2 -17128.013} C_VEL
LIN {X 0,Y 284.268,Z 234.072,A -85,B 0,C 180,E1 -17131.277,E2 -17131.277} C_VEL
LIN {X 0,Y 284.317,Z 234.063,A -85,B 0,C 180,E1 -17135.35,E2 -17135.35} C_VEL
LIN {X 0,Y 284.304,Z 234.064,A -85,B 0,C 180,E1 -17138.17,E2 -17138.17} C_VEL
LIN {X 0,Y 284.307,Z 234.066,A -85,B 0,C 180,E1 -17142.14,E2 -17142.14} C_VEL
LIN {X 0,Y 284.251,Z 234.078,A -85,B 0,C 180,E1 -17146.195,E2 -17146.195} C_VEL
LIN {X 0,Y 284.292,Z 234.074,A -85,B 0,C 180,E1 -17150.027,E2 -17150.027} C_VEL
LIN {X 0,Y 284.322,Z 234.067,A -85,B 0,C 180,E1 -17153.617,E2 -17153.617} C_VEL
LIN {X 0,Y 284.296,Z 234.064,A -85,B 0,C 180,E1 -17157.193,E2 -17157.193} C_VEL
LIN {X 0,Y 284.351,Z 234.061,A -85,B 0,C 180,E1 -17160.379,E2 -17160.379} C_VEL
LIN {X 0,Y 284.37,Z 234.063,A -85,B 0,C 180,E1 -17163.589,E2 -17163.589} C_VEL
LIN {X 0,Y 284.36,Z 234.061,A -85,B 0,C 180,E1 -17166.709,E2 -17166.709} C_VEL
LIN {X 0,Y 284.398,Z 234.055,A -85,B 0,C 180,E1 -17171.264,E2 -17171.264} C_VEL
LIN {X 0,Y 284.488,Z 234.045,A -85,B 0,C 180,E1 -17174.461,E2 -17174.461} C_VEL
LIN {X 0,Y 284.485,Z 234.045,A -85,B 0,C 180,E1 -17178.603,E2 -17178.603} C_VEL
LIN {X 0,Y 284.655,Z 234.028,A -85,B 0,C 180,E1 -17181.482,E2 -17181.482} C_VEL
LIN {X 0,Y 284.597,Z 234.032,A -85,B 0,C 180,E1 -17184.332,E2 -17184.332} C_VEL
LIN {X 0,Y 284.854,Z 234,A -85,B 0,C 180,E1 -17188.587,E2 -17188.587} C_VEL
LIN {X 0,Y 284.853,Z 234.002,A -85,B 0,C 180,E1 -17191.414,E2 -17191.414} C_VEL
LIN {X 0,Y 284.687,Z 234.025,A -85,B 0,C 180,E1 -17197.09,E2 -17197.09} C_VEL
LIN {X 0,Y 284.519,Z 234.042,A -85,B 0,C 180,E1 -17199.956,E2 -17199.956} C_VEL
LIN {X 0,Y 284.478,Z 234.049,A -85,B 0,C 180,E1 -17204.301,E2 -17204.301} C_VEL
LIN {X 0,Y 284.418,Z 234.057,A -85,B 0,C 180,E1 -17207.247,E2 -17207.247} C_VEL
LIN {X 0,Y 284.372,Z 234.061,A -85,B 0,C 180,E1 -17210.24,E2 -17210.24} C_VEL
LIN {X 0,Y 284.411,Z 234.196,A -85,B 0,C 180,E1 -17213.618,E2 -17213.618} C_VEL
LIN {X 0,Y 293.316,Z 259.147,A -85,B 0,C 180,E1 -17215.036,E2 -17215.036} C_VEL
LIN {X 0,Y 295.211,Z 264.723,A -85,B 0,C 180,E1 -17215.335,E2 -17215.335} C_VEL
LIN {X 0,Y 292.703,Z 341.337,A -85,B 0,C 180,E1 -17217.474,E2 -17217.474} C_VEL
LIN {X 0,Y 291.937,Z 355.172,A -85,B 0,C 180,E1 -17218.139,E2 -17218.139} C_VEL
LIN {X 0,Y 291.137,Z 367.402,A -85,B 0,C 180,E1 -17218.998,E2 -17218.998} C_VEL
LIN {X 0,Y 290.019,Z 379.772,A -85,B 0,C 180,E1 -17220.166,E2 -17220.166} C_VEL
LIN {X 0,Y 288.743,Z 391.436,A -85,B 0,C 180,E1 -17221.582,E2 -17221.582} C_VEL
LIN {X 0,Y 287.592,Z 401.209,A -85,B 0,C 180,E1 -17223.066,E2 -17223.066} C_VEL
LIN {X 0,Y 286.227,Z 411.532,A -85,B 0,C 180,E1 -17225.022,E2 -17225.022} C_VEL
LIN {X 0,Y 285.09,Z 419.973,A -85,B 0,C 180,E1 -17227.008,E2 -17227.008} C_VEL
LIN {X 0,Y 284.187,Z 426.818,A -85,B 0,C 180,E1 -17229.004,E2 -17229.004} C_VEL
LIN {X 0,Y 283.384,Z 433.372,A -85,B 0,C 180,E1 -17231.441,E2 -17231.441} C_VEL
LIN {X 0,Y 282.87,Z 438.399,A -85,B 0,C 180,E1 -17233.904,E2 -17233.904} C_VEL
LIN {X 0,Y 282.423,Z 441.764,A -85,B 0,C 180,E1 -17236.185,E2 -17236.185} C_VEL
LIN {X 0,Y 282.254,Z 443.867,A -85,B 0,C 180,E1 -17238.323,E2 -17238.323} C_VEL
LIN {X 0,Y 282.215,Z 445.055,A -85,B 0,C 180,E1 -17240.526,E2 -17240.526} C_VEL
LIN {X 0,Y 282.473,Z 445.153,A -85,B 0,C 180,E1 -17243.336,E2 -17243.336} C_VEL
LIN {X 0,Y 282.784,Z 444.402,A -85,B 0,C 180,E1 -17245.138,E2 -17245.138} C_VEL
LIN {X 0,Y 283.47,Z 442.456,A -85,B 0,C 180,E1 -17247.443,E2 -17247.443} C_VEL
LIN {X 0,Y 284.439,Z 439.197,A -85,B 0,C 180,E1 -17249.848,E2 -17249.848} C_VEL
LIN {X 0,Y 285.711,Z 434.464,A -85,B 0,C 180,E1 -17252.306,E2 -17252.306} C_VEL
LIN {X 0,Y 287.393,Z 428.071,A -85,B 0,C 180,E1 -17254.784,E2 -17254.784} C_VEL
LIN {X 0,Y 289.093,Z 421.59,A -85,B 0,C 180,E1 -17256.732,E2 -17256.732} C_VEL
LIN {X 0,Y 291.066,Z 413.143,A -85,B 0,C 180,E1 -17258.766,E2 -17258.766} C_VEL
LIN {X 0,Y 293.132,Z 403.783,A -85,B 0,C 180,E1 -17260.57,E2 -17260.57} C_VEL
LIN {X 0,Y 295.277,Z 393.342,A -85,B 0,C 180,E1 -17262.167,E2 -17262.167} C_VEL
LIN {X 0,Y 297.221,Z 382.247,A -85,B 0,C 180,E1 -17263.516,E2 -17263.516} C_VEL
LIN {X 0,Y 298.937,Z 370.416,A -85,B 0,C 180,E1 -17264.647,E2 -17264.647} C_VEL
LIN {X 0,Y 300.35,Z 357.237,A -85,B 0,C 180,E1 -17265.583,E2 -17265.583} C_VEL
LIN {X 0,Y 301.215,Z 346.903,A -85,B 0,C 180,E1 -17266.105,E2 -17266.105} C_VEL
LIN {X 0,Y 300.974,Z 341.196,A -85,B 0,C 180,E1 -17266.401,E2 -17266.401} C_VEL
LIN {X 0,Y 297.117,Z 322.738,A -85,B 0,C 180,E1 -17267.577,E2 -17267.577} C_VEL
LIN {X 0,Y 296.873,Z 316.968,A -85,B 0,C 180,E1 -17267.811,E2 -17267.811} C_VEL
LIN {X 0,Y 299.076,Z 275.695,A -85,B 0,C 180,E1 -17269.008,E2 -17269.008} C_VEL
LIN {X 0,Y 293.18,Z 262.836,A -85,B 0,C 180,E1 -17270.412,E2 -17270.412} C_VEL
LIN {X 0,Y 287.26,Z 251.942,A -85,B 0,C 180,E1 -17271.869,E2 -17271.869} C_VEL
LIN {X 0,Y 283.086,Z 244.99,A -85,B 0,C 180,E1 -17272.942,E2 -17272.942} C_VEL
LIN {X 0,Y 280.723,Z 241.213,A -85,B 0,C 180,E1 -17273.576,E2 -17273.576} C_VEL
LIN {X 0,Y 278.27,Z 237.293,A -85,B 0,C 180,E1 -17274.293,E2 -17274.293} C_VEL
LIN {X 0,Y 277.44,Z 234.926,A -85,B 0,C 180,E1 -17275.551,E2 -17275.551} C_VEL
LIN {X 0,Y 277.784,Z 234.882,A -85,B 0,C 180,E1 -17278.551,E2 -17278.551} C_VEL
LIN {X 0,Y 277.783,Z 234.882,A -85,B 0,C 180,E1 -17281.45,E2 -17281.45} C_VEL
LIN {X 0,Y 277.596,Z 234.908,A -85,B 0,C 180,E1 -17287.273,E2 -17287.273} C_VEL
LIN {X 0,Y 277.429,Z 234.928,A -85,B 0,C 180,E1 -17290.215,E2 -17290.215} C_VEL
LIN {X 0,Y 277.378,Z 234.927,A -85,B 0,C 180,E1 -17294.678,E2 -17294.678} C_VEL
LIN {X 0,Y 277.257,Z 234.948,A -85,B 0,C 180,E1 -17299.241,E2 -17299.241} C_VEL
LIN {X 0,Y 277.267,Z 234.94,A -85,B 0,C 180,E1 -17303.927,E2 -17303.927} C_VEL
LIN {X 0,Y 277.284,Z 234.942,A -85,B 0,C 180,E1 -17307.5,E2 -17307.5} C_VEL
LIN {X 0,Y 277.227,Z 234.948,A -85,B 0,C 180,E1 -17310.476,E2 -17310.476} C_VEL
LIN {X 0,Y 277.218,Z 234.953,A -85,B 0,C 180,E1 -17313.9,E2 -17313.9} C_VEL
LIN {X 0,Y 277.244,Z 234.948,A -85,B 0,C 180,E1 -17317.474,E2 -17317.474} C_VEL
LIN {X 0,Y 277.192,Z 234.953,A -85,B 0,C 180,E1 -17321.24,E2 -17321.24} C_VEL
LIN {X 0,Y 277.187,Z 234.953,A -85,B 0,C 180,E1 -17325.23,E2 -17325.23} C_VEL
LIN {X 0,Y 277.232,Z 235.008,A -85,B 0,C 180,E1 -17328.414,E2 -17328.414} C_VEL
LIN {X 0,Y 279.638,Z 242.522,A -85,B 0,C 180,E1 -17331.917,E2 -17331.917} C_VEL
LIN {X 0,Y 281.937,Z 250.852,A -85,B 0,C 180,E1 -17335.348,E2 -17335.348} C_VEL
LIN {X 0,Y 282.853,Z 254.488,A -85,B 0,C 180,E1 -17336.713,E2 -17336.713} C_VEL
LIN {X 0,Y 285.393,Z 259.338,A -85,B 0,C 180,E1 -17337.393,E2 -17337.393} C_VEL
LIN {X 0,Y 291.016,Z 271.118,A -85,B 0,C 180,E1 -17338.853,E2 -17338.853} C_VEL
LIN {X 0,Y 292.999,Z 276.054,A -85,B 0,C 180,E1 -17339.362,E2 -17339.362} C_VEL
LIN {X 0,Y 296.022,Z 294.025,A -85,B 0,C 180,E1 -17340.511,E2 -17340.511} C_VEL
LIN {X 0,Y 297.672,Z 308.061,A -85,B 0,C 180,E1 -17341.274,E2 -17341.274} C_VEL
LIN {X 0,Y 294.717,Z 366.343,A -85,B 0,C 180,E1 -17342.994,E2 -17342.994} C_VEL
LIN {X 0,Y 293.381,Z 380.598,A -85,B 0,C 180,E1 -17343.697,E2 -17343.697} C_VEL
LIN {X 0,Y 291.635,Z 392.163,A -85,B 0,C 180,E1 -17344.487,E2 -17344.487} C_VEL
LIN {X 0,Y 289.537,Z 404.429,A -85,B 0,C 180,E1 -17345.632,E2 -17345.632} C_VEL
LIN {X 0,Y 287.344,Z 415.54,A -85,B 0,C 180,E1 -17346.965,E2 -17346.965} C_VEL
LIN {X 0,Y 285.076,Z 425.683,A -85,B 0,C 180,E1 -17348.489,E2 -17348.489} C_VEL
LIN {X 0,Y 282.668,Z 435.739,A -85,B 0,C 180,E1 -17350.39,E2 -17350.39} C_VEL
LIN {X 0,Y 280.523,Z 444.68,A -85,B 0,C 180,E1 -17352.506,E2 -17352.506} C_VEL
LIN {X 0,Y 278.821,Z 451.873,A -85,B 0,C 180,E1 -17354.655,E2 -17354.655} C_VEL
LIN {X 0,Y 277.271,Z 457.671,A -85,B 0,C 180,E1 -17356.815,E2 -17356.815} C_VEL
LIN {X 0,Y 276.336,Z 462.271,A -85,B 0,C 180,E1 -17359.005,E2 -17359.005} C_VEL
LIN {X 0,Y 275.712,Z 465.794,A -85,B 0,C 180,E1 -17361.203,E2 -17361.203} C_VEL
LIN {X 0,Y 275.452,Z 467.578,A -85,B 0,C 180,E1 -17362.671,E2 -17362.671} C_VEL
LIN {X 0,Y 275.287,Z 469.346,A -85,B 0,C 180,E1 -17364.665,E2 -17364.665} C_VEL
LIN {X 0,Y 275.346,Z 470.444,A -85,B 0,C 180,E1 -17367.074,E2 -17367.074} C_VEL
LIN {X 0,Y 275.35,Z 470.555,A -85,B 0,C 180,E1 -17368.537,E2 -17368.537} C_VEL
LIN {X 0,Y 275.415,Z 470.267,A -85,B 0,C 180,E1 -17370,E2 -17370} C_VEL
LIN {X 0,Y 275.374,Z 469.555,A -85,B 0,C 180,E1 -17371.462,E2 -17371.462} C_VEL
LIN {X 0,Y 275.383,Z 468.375,A -85,B 0,C 180,E1 -17372.925,E2 -17372.925} C_VEL
LIN {X 0,Y 275.43,Z 465.024,A -85,B 0,C 180,E1 -17375.645,E2 -17375.645} C_VEL
LIN {X 0,Y 275.588,Z 460.668,A -85,B 0,C 180,E1 -17378.062,E2 -17378.062} C_VEL
LIN {X 0,Y 276.093,Z 454.379,A -85,B 0,C 180,E1 -17380.634,E2 -17380.634} C_VEL
LIN {X 0,Y 276.857,Z 447.479,A -85,B 0,C 180,E1 -17382.832,E2 -17382.832} C_VEL
LIN {X 0,Y 277.969,Z 438.863,A -85,B 0,C 180,E1 -17385.018,E2 -17385.018} C_VEL
LIN {X 0,Y 279.056,Z 430.372,A -85,B 0,C 180,E1 -17386.755,E2 -17386.755} C_VEL
LIN {X 0,Y 280.4,Z 420.206,A -85,B 0,C 180,E1 -17388.445,E2 -17388.445} C_VEL
LIN {X 0,Y 281.794,Z 409.595,A -85,B 0,C 180,E1 -17389.863,E2 -17389.863} C_VEL
LIN {X 0,Y 283.104,Z 397.852,A -85,B 0,C 180,E1 -17391.095,E2 -17391.095} C_VEL
LIN {X 0,Y 284.295,Z 385.844,A -85,B 0,C 180,E1 -17392.049,E2 -17392.049} C_VEL
LIN {X 0,Y 285.279,Z 373.105,A -85,B 0,C 180,E1 -17392.78,E2 -17392.78} C_VEL
LIN {X 0,Y 285.996,Z 359.058,A -85,B 0,C 180,E1 -17393.28,E2 -17393.28} C_VEL
LIN {X 0,Y 287.454,Z 304.152,A -85,B 0,C 180,E1 -17394.861,E2 -17394.861} C_VEL
LIN {X 0,Y 281.754,Z 258.706,A -85,B 0,C 180,E1 -17396.725,E2 -17396.725} C_VEL
LIN {X 0,Y 281.416,Z 254.746,A -85,B 0,C 180,E1 -17397.918,E2 -17397.918} C_VEL
LIN {X 0,Y 279.123,Z 243.55,A -85,B 0,C 180,E1 -17401.45,E2 -17401.45} C_VEL
LIN {X 0,Y 277.298,Z 234.945,A -85,B 0,C 180,E1 -17404.323,E2 -17404.323} C_VEL
LIN {X 0,Y 277.247,Z 234.951,A -85,B 0,C 180,E1 -17408.202,E2 -17408.202} C_VEL
LIN {X 0,Y 277.201,Z 234.955,A -85,B 0,C 180,E1 -17412.671,E2 -17412.671} C_VEL
LIN {X 0,Y 277.193,Z 234.956,A -85,B 0,C 180,E1 -17416.798,E2 -17416.798} C_VEL
LIN {X 0,Y 277.216,Z 234.952,A -85,B 0,C 180,E1 -17420.668,E2 -17420.668} C_VEL
LIN {X 0,Y 277.262,Z 234.945,A -85,B 0,C 180,E1 -17424.338,E2 -17424.338} C_VEL
LIN {X 0,Y 277.206,Z 234.955,A -85,B 0,C 180,E1 -17427.831,E2 -17427.831} C_VEL
LIN {X 0,Y 277.23,Z 234.952,A -85,B 0,C 180,E1 -17431.205,E2 -17431.205} C_VEL
LIN {X 0,Y 277.273,Z 234.942,A -85,B 0,C 180,E1 -17434.475,E2 -17434.475} C_VEL
LIN {X 0,Y 277.232,Z 234.952,A -85,B 0,C 180,E1 -17437.65,E2 -17437.65} C_VEL
LIN {X 0,Y 277.254,Z 234.947,A -85,B 0,C 180,E1 -17440.759,E2 -17440.759} C_VEL
LIN {X 0,Y 277.377,Z 234.931,A -85,B 0,C 180,E1 -17445.322,E2 -17445.322} C_VEL
LIN {X 0,Y 277.428,Z 234.925,A -85,B 0,C 180,E1 -17449.785,E2 -17449.785} C_VEL
LIN {X 0,Y 277.599,Z 234.906,A -85,B 0,C 180,E1 -17452.727,E2 -17452.727} C_VEL
LIN {X 0,Y 277.782,Z 234.875,A -85,B 0,C 180,E1 -17458.55,E2 -17458.55} C_VEL
LIN {X 0,Y 277.783,Z 234.876,A -85,B 0,C 180,E1 -17461.449,E2 -17461.449} C_VEL
LIN {X 0,Y 277.603,Z 234.904,A -85,B 0,C 180,E1 -17467.272,E2 -17467.272} C_VEL
LIN {X 0,Y 277.427,Z 234.926,A -85,B 0,C 180,E1 -17470.214,E2 -17470.214} C_VEL
LIN {X 0,Y 277.383,Z 234.928,A -85,B 0,C 180,E1 -17474.676,E2 -17474.676} C_VEL
LIN {X 0,Y 277.34,Z 234.925,A -85,B 0,C 180,E1 -17479.234,E2 -17479.234} C_VEL
LIN {X 0,Y 277.348,Z 234.932,A -85,B 0,C 180,E1 -17483.918,E2 -17483.918} C_VEL
LIN {X 0,Y 277.298,Z 234.941,A -85,B 0,C 180,E1 -17487.506,E2 -17487.506} C_VEL
LIN {X 0,Y 277.248,Z 234.95,A -85,B 0,C 180,E1 -17490.484,E2 -17490.484} C_VEL
LIN {X 0,Y 277.222,Z 234.95,A -85,B 0,C 180,E1 -17493.899,E2 -17493.899} C_VEL
LIN {X 0,Y 277.254,Z 234.939,A -85,B 0,C 180,E1 -17497.471,E2 -17497.471} C_VEL
LIN {X 0,Y 277.237,Z 234.94,A -85,B 0,C 180,E1 -17501.231,E2 -17501.231} C_VEL
LIN {X 0,Y 277.205,Z 234.95,A -85,B 0,C 180,E1 -17505.225,E2 -17505.225} C_VEL
LIN {X 0,Y 277.208,Z 234.954,A -85,B 0,C 180,E1 -17509.515,E2 -17509.515} C_VEL
LIN {X 0,Y 277.259,Z 234.945,A -85,B 0,C 180,E1 -17512.534,E2 -17512.534} C_VEL
LIN {X 0,Y 277.235,Z 234.944,A -85,B 0,C 180,E1 -17516.107,E2 -17516.107} C_VEL
LIN {X 0,Y 277.251,Z 234.944,A -85,B 0,C 180,E1 -17519.541,E2 -17519.541} C_VEL
LIN {X 0,Y 277.351,Z 234.934,A -85,B 0,C 180,E1 -17522.867,E2 -17522.867} C_VEL
LIN {X 0,Y 277.322,Z 234.94,A -85,B 0,C 180,E1 -17526.082,E2 -17526.082} C_VEL
LIN {X 0,Y 277.34,Z 234.932,A -85,B 0,C 180,E1 -17530.768,E2 -17530.768} C_VEL
LIN {X 0,Y 277.431,Z 234.927,A -85,B 0,C 180,E1 -17535.327,E2 -17535.327} C_VEL
LIN {X 0,Y 277.504,Z 234.914,A -85,B 0,C 180,E1 -17539.79,E2 -17539.79} C_VEL
LIN {X 0,Y 277.647,Z 234.898,A -85,B 0,C 180,E1 -17542.73,E2 -17542.73} C_VEL
LIN {X 0,Y 277.82,Z 234.876,A -85,B 0,C 180,E1 -17548.551,E2 -17548.551} C_VEL
LIN {X 0,Y 277.819,Z 234.878,A -85,B 0,C 180,E1 -17551.45,E2 -17551.45} C_VEL
LIN {X 0,Y 277.642,Z 234.903,A -85,B 0,C 180,E1 -17557.271,E2 -17557.271} C_VEL
LIN {X 0,Y 277.46,Z 234.922,A -85,B 0,C 180,E1 -17560.212,E2 -17560.212} C_VEL
LIN {X 0,Y 277.431,Z 234.929,A -85,B 0,C 180,E1 -17564.673,E2 -17564.673} C_VEL
LIN {X 0,Y 277.337,Z 234.939,A -85,B 0,C 180,E1 -17569.232,E2 -17569.232} C_VEL
LIN {X 0,Y 277.304,Z 234.944,A -85,B 0,C 180,E1 -17573.079,E2 -17573.079} C_VEL
LIN {X 0,Y 286.017,Z 258.763,A -85,B 0,C 180,E1 -17574.512,E2 -17574.512} C_VEL
LIN {X 0,Y 288.376,Z 265.902,A -85,B 0,C 180,E1 -17574.9,E2 -17574.9} C_VEL
LIN {X 0,Y 285.851,Z 342.753,A -85,B 0,C 180,E1 -17577.126,E2 -17577.126} C_VEL
LIN {X 0,Y 285.061,Z 356.412,A -85,B 0,C 180,E1 -17577.817,E2 -17577.817} C_VEL
LIN {X 0,Y 284.21,Z 368.694,A -85,B 0,C 180,E1 -17578.725,E2 -17578.725} C_VEL
LIN {X 0,Y 282.988,Z 381.42,A -85,B 0,C 180,E1 -17579.984,E2 -17579.984} C_VEL
LIN {X 0,Y 281.774,Z 392.39,A -85,B 0,C 180,E1 -17581.373,E2 -17581.373} C_VEL
LIN {X 0,Y 280.442,Z 402.979,A -85,B 0,C 180,E1 -17583.063,E2 -17583.063} C_VEL
LIN {X 0,Y 279.087,Z 412.94,A -85,B 0,C 180,E1 -17585.041,E2 -17585.041} C_VEL
LIN {X 0,Y 277.927,Z 421.058,A -85,B 0,C 180,E1 -17587.046,E2 -17587.046} C_VEL
LIN {X 0,Y 276.954,Z 428.533,A -85,B 0,C 180,E1 -17589.37,E2 -17589.37} C_VEL
LIN {X 0,Y 276.178,Z 434.884,A -85,B 0,C 180,E1 -17591.9,E2 -17591.9} C_VEL
LIN {X 0,Y 275.661,Z 439.607,A -85,B 0,C 180,E1 -17594.451,E2 -17594.451} C_VEL
LIN {X 0,Y 275.29,Z 442.309,A -85,B 0,C 180,E1 -17596.426,E2 -17596.426} C_VEL
LIN {X 0,Y 275.154,Z 444.166,A -85,B 0,C 180,E1 -17598.388,E2 -17598.388} C_VEL
LIN {X 0,Y 275.135,Z 445.25,A -85,B 0,C 180,E1 -17600.314,E2 -17600.314} C_VEL
LIN {X 0,Y 275.263,Z 445.65,A -85,B 0,C 180,E1 -17602.317,E2 -17602.317} C_VEL
LIN {X 0,Y 275.618,Z 445.126,A -85,B 0,C 180,E1 -17604.674,E2 -17604.674} C_VEL
LIN {X 0,Y 276.238,Z 443.489,A -85,B 0,C 180,E1 -17607.086,E2 -17607.086} C_VEL
LIN {X 0,Y 277.204,Z 440.638,A -85,B 0,C 180,E1 -17609.532,E2 -17609.532} C_VEL
LIN {X 0,Y 278.472,Z 436.394,A -85,B 0,C 180,E1 -17612.034,E2 -17612.034} C_VEL
LIN {X 0,Y 280.143,Z 430.518,A -85,B 0,C 180,E1 -17614.56,E2 -17614.56} C_VEL
LIN {X 0,Y 282.109,Z 423.507,A -85,B 0,C 180,E1 -17616.851,E2 -17616.851} C_VEL
LIN {X 0,Y 284.189,Z 415.303,A -85,B 0,C 180,E1 -17618.979,E2 -17618.979} C_VEL
LIN {X 0,Y 286.288,Z 406.341,A -85,B 0,C 180,E1 -17620.833,E2 -17620.833} C_VEL
LIN {X 0,Y 288.724,Z 395.518,A -85,B 0,C 180,E1 -17622.599,E2 -17622.599} C_VEL
LIN {X 0,Y 290.686,Z 385.311,A -85,B 0,C 180,E1 -17623.929,E2 -17623.929} C_VEL
LIN {X 0,Y 292.538,Z 373.67,A -85,B 0,C 180,E1 -17625.123,E2 -17625.123} C_VEL
LIN {X 0,Y 294.093,Z 361.324,A -85,B 0,C 180,E1 -17626.087,E2 -17626.087} C_VEL
LIN {X 0,Y 295.199,Z 349.203,A -85,B 0,C 180,E1 -17626.776,E2 -17626.776} C_VEL
LIN {X 0,Y 295.977,Z 335.984,A -85,B 0,C 180,E1 -17627.256,E2 -17627.256} C_VEL
LIN {X 0,Y 296.873,Z 316.968,A -85,B 0,C 180,E1 -17627.811,E2 -17627.811} C_VEL
LIN {X 0,Y 296.646,Z 311.197,A -85,B 0,C 180,E1 -17628.054,E2 -17628.054} C_VEL
LIN {X 0,Y 293.094,Z 292.714,A -85,B 0,C 180,E1 -17629.277,E2 -17629.277} C_VEL
LIN {X 0,Y 292.926,Z 286.945,A -85,B 0,C 180,E1 -17629.524,E2 -17629.524} C_VEL
LIN {X 0,Y 293.311,Z 277.782,A -85,B 0,C 180,E1 -17629.816,E2 -17629.816} C_VEL
LIN {X 0,Y 287.783,Z 265.742,A -85,B 0,C 180,E1 -17631.208,E2 -17631.208} C_VEL
LIN {X 0,Y 281.376,Z 253.917,A -85,B 0,C 180,E1 -17632.883,E2 -17632.883} C_VEL
LIN {X 0,Y 276.541,Z 246.147,A -85,B 0,C 180,E1 -17634.216,E2 -17634.216} C_VEL
LIN {X 0,Y 273.947,Z 242.28,A -85,B 0,C 180,E1 -17634.964,E2 -17634.964} C_VEL
LIN {X 0,Y 270.989,Z 237.861,A -85,B 0,C 180,E1 -17635.911,E2 -17635.911} C_VEL
LIN {X 0,Y 270.591,Z 235.778,A -85,B 0,C 180,E1 -17637.023,E2 -17637.023} C_VEL
LIN {X 0,Y 270.788,Z 235.757,A -85,B 0,C 180,E1 -17640.001,E2 -17640.001} C_VEL
LIN {X 0,Y 270.588,Z 235.777,A -85,B 0,C 180,E1 -17642.978,E2 -17642.978} C_VEL
LIN {X 0,Y 270.554,Z 235.784,A -85,B 0,C 180,E1 -17647.463,E2 -17647.463} C_VEL
LIN {X 0,Y 270.381,Z 235.803,A -85,B 0,C 180,E1 -17650.484,E2 -17650.484} C_VEL
LIN {X 0,Y 270.338,Z 235.806,A -85,B 0,C 180,E1 -17655.069,E2 -17655.069} C_VEL
LIN {X 0,Y 270.196,Z 235.824,A -85,B 0,C 180,E1 -17659.764,E2 -17659.764} C_VEL
LIN {X 0,Y 270.211,Z 235.823,A -85,B 0,C 180,E1 -17664.592,E2 -17664.592} C_VEL
LIN {X 0,Y 270.22,Z 235.824,A -85,B 0,C 180,E1 -17667.915,E2 -17667.915} C_VEL
LIN {X 0,Y 270.148,Z 235.834,A -85,B 0,C 180,E1 -17671.354,E2 -17671.354} C_VEL
LIN {X 0,Y 270.178,Z 235.825,A -85,B 0,C 180,E1 -17674.91,E2 -17674.91} C_VEL
LIN {X 0,Y 270.181,Z 235.827,A -85,B 0,C 180,E1 -17678.714,E2 -17678.714} C_VEL
LIN {X 0,Y 270.15,Z 235.829,A -85,B 0,C 180,E1 -17683.252,E2 -17683.252} C_VEL
LIN {X 0,Y 270.154,Z 235.881,A -85,B 0,C 180,E1 -17686.896,E2 -17686.896} C_VEL
LIN {X 0,Y 272.628,Z 243.317,A -85,B 0,C 180,E1 -17690.657,E2 -17690.657} C_VEL
LIN {X 0,Y 274.777,Z 250.786,A -85,B 0,C 180,E1 -17693.97,E2 -17693.97} C_VEL
LIN {X 0,Y 275.65,Z 254.103,A -85,B 0,C 180,E1 -17695.25,E2 -17695.25} C_VEL
LIN {X 0,Y 281.535,Z 265.271,A -85,B 0,C 180,E1 -17696.93,E2 -17696.93} C_VEL
LIN {X 0,Y 286.111,Z 274.917,A -85,B 0,C 180,E1 -17698.166,E2 -17698.166} C_VEL
LIN {X 0,Y 287.828,Z 279.321,A -85,B 0,C 180,E1 -17698.643,E2 -17698.643} C_VEL
LIN {X 0,Y 290.688,Z 297.411,A -85,B 0,C 180,E1 -17699.818,E2 -17699.818} C_VEL
LIN {X 0,Y 291.969,Z 309.187,A -85,B 0,C 180,E1 -17700.466,E2 -17700.466} C_VEL
LIN {X 0,Y 288.894,Z 366.021,A -85,B 0,C 180,E1 -17702.194,E2 -17702.194} C_VEL
LIN {X 0,Y 287.442,Z 380.369,A -85,B 0,C 180,E1 -17702.913,E2 -17702.913} C_VEL
LIN {X 0,Y 285.652,Z 391.881,A -85,B 0,C 180,E1 -17703.716,E2 -17703.716} C_VEL
LIN {X 0,Y 283.447,Z 404.137,A -85,B 0,C 180,E1 -17704.877,E2 -17704.877} C_VEL
LIN {X 0,Y 281.156,Z 415.24,A -85,B 0,C 180,E1 -17706.232,E2 -17706.232} C_VEL
LIN {X 0,Y 278.801,Z 425.371,A -85,B 0,C 180,E1 -17707.785,E2 -17707.785} C_VEL
LIN {X 0,Y 276.405,Z 434.581,A -85,B 0,C 180,E1 -17709.539,E2 -17709.539} C_VEL
LIN {X 0,Y 274.036,Z 443.987,A -85,B 0,C 180,E1 -17711.798,E2 -17711.798} C_VEL
LIN {X 0,Y 271.986,Z 452.002,A -85,B 0,C 180,E1 -17714.259,E2 -17714.259} C_VEL
LIN {X 0,Y 270.354,Z 457.711,A -85,B 0,C 180,E1 -17716.471,E2 -17716.471} C_VEL
LIN {X 0,Y 269.333,Z 462.226,A -85,B 0,C 180,E1 -17718.715,E2 -17718.715} C_VEL
LIN {X 0,Y 268.675,Z 465.67,A -85,B 0,C 180,E1 -17720.971,E2 -17720.971} C_VEL
LIN {X 0,Y 268.222,Z 468.746,A -85,B 0,C 180,E1 -17723.984,E2 -17723.984} C_VEL
LIN {X 0,Y 268.168,Z 469.644,A -85,B 0,C 180,E1 -17725.491,E2 -17725.491} C_VEL
LIN {X 0,Y 268.249,Z 470.126,A -85,B 0,C 180,E1 -17726.997,E2 -17726.997} C_VEL
LIN {X 0,Y 268.273,Z 470.204,A -85,B 0,C 180,E1 -17728.499,E2 -17728.499} C_VEL
LIN {X 0,Y 268.332,Z 469.88,A -85,B 0,C 180,E1 -17730,E2 -17730} C_VEL
LIN {X 0,Y 268.296,Z 469.1,A -85,B 0,C 180,E1 -17731.501,E2 -17731.501} C_VEL
LIN {X 0,Y 268.312,Z 467.88,A -85,B 0,C 180,E1 -17733.002,E2 -17733.002} C_VEL
LIN {X 0,Y 268.361,Z 464.685,A -85,B 0,C 180,E1 -17735.631,E2 -17735.631} C_VEL
LIN {X 0,Y 268.525,Z 459.981,A -85,B 0,C 180,E1 -17738.275,E2 -17738.275} C_VEL
LIN {X 0,Y 269.062,Z 453.576,A -85,B 0,C 180,E1 -17740.915,E2 -17740.915} C_VEL
LIN {X 0,Y 269.922,Z 446.574,A -85,B 0,C 180,E1 -17743.167,E2 -17743.167} C_VEL
LIN {X 0,Y 270.817,Z 439.389,A -85,B 0,C 180,E1 -17745.039,E2 -17745.039} C_VEL
LIN {X 0,Y 272.082,Z 430.089,A -85,B 0,C 180,E1 -17747.009,E2 -17747.009} C_VEL
LIN {X 0,Y 273.451,Z 419.955,A -85,B 0,C 180,E1 -17748.737,E2 -17748.737} C_VEL
LIN {X 0,Y 274.883,Z 409.357,A -85,B 0,C 180,E1 -17750.189,E2 -17750.189} C_VEL
LIN {X 0,Y 276.235,Z 397.648,A -85,B 0,C 180,E1 -17751.45,E2 -17751.45} C_VEL
LIN {X 0,Y 277.606,Z 384.432,A -85,B 0,C 180,E1 -17752.511,E2 -17752.511} C_VEL
LIN {X 0,Y 278.6,Z 371.117,A -85,B 0,C 180,E1 -17753.26,E2 -17753.26} C_VEL
LIN {X 0,Y 279.311,Z 354.729,A -85,B 0,C 180,E1 -17753.815,E2 -17753.815} C_VEL
LIN {X 0,Y 280.77,Z 305.298,A -85,B 0,C 180,E1 -17755.27,E2 -17755.27} C_VEL
LIN {X 0,Y 274.827,Z 258.46,A -85,B 0,C 180,E1 -17757.247,E2 -17757.247} C_VEL
LIN {X 0,Y 272.831,Z 248.055,A -85,B 0,C 180,E1 -17760.577,E2 -17760.577} C_VEL
LIN {X 0,Y 270.498,Z 237.044,A -85,B 0,C 180,E1 -17764.255,E2 -17764.255} C_VEL
LIN {X 0,Y 270.237,Z 235.823,A -85,B 0,C 180,E1 -17764.744,E2 -17764.744} C_VEL
LIN {X 0,Y 270.187,Z 235.828,A -85,B 0,C 180,E1 -17768.707,E2 -17768.707} C_VEL
LIN {X 0,Y 270.151,Z 235.834,A -85,B 0,C 180,E1 -17773.245,E2 -17773.245} C_VEL
LIN {X 0,Y 270.155,Z 235.835,A -85,B 0,C 180,E1 -17777.438,E2 -17777.438} C_VEL
LIN {X 0,Y 270.19,Z 235.829,A -85,B 0,C 180,E1 -17781.371,E2 -17781.371} C_VEL
LIN {X 0,Y 270.177,Z 235.828,A -85,B 0,C 180,E1 -17785.09,E2 -17785.09} C_VEL
LIN {X 0,Y 270.161,Z 235.832,A -85,B 0,C 180,E1 -17789.134,E2 -17789.134} C_VEL
LIN {X 0,Y 270.236,Z 235.819,A -85,B 0,C 180,E1 -17792.145,E2 -17792.145} C_VEL
LIN {X 0,Y 270.21,Z 235.827,A -85,B 0,C 180,E1 -17795.537,E2 -17795.537} C_VEL
LIN {X 0,Y 270.194,Z 235.825,A -85,B 0,C 180,E1 -17800.236,E2 -17800.236} C_VEL
LIN {X 0,Y 270.337,Z 235.804,A -85,B 0,C 180,E1 -17804.931,E2 -17804.931} C_VEL
LIN {X 0,Y 270.38,Z 235.805,A -85,B 0,C 180,E1 -17809.516,E2 -17809.516} C_VEL
LIN {X 0,Y 270.556,Z 235.782,A -85,B 0,C 180,E1 -17812.537,E2 -17812.537} C_VEL
LIN {X 0,Y 270.748,Z 235.75,A -85,B 0,C 180,E1 -17818.512,E2 -17818.512} C_VEL
LIN {X 0,Y 270.75,Z 235.752,A -85,B 0,C 180,E1 -17821.487,E2 -17821.487} C_VEL
LIN {X 0,Y 270.559,Z 235.781,A -85,B 0,C 180,E1 -17827.462,E2 -17827.462} C_VEL
LIN {X 0,Y 270.38,Z 235.805,A -85,B 0,C 180,E1 -17830.483,E2 -17830.483} C_VEL
LIN {X 0,Y 270.351,Z 235.8,A -85,B 0,C 180,E1 -17835.067,E2 -17835.067} C_VEL
LIN {X 0,Y 270.298,Z 235.8,A -85,B 0,C 180,E1 -17839.755,E2 -17839.755} C_VEL
LIN {X 0,Y 270.262,Z 235.819,A -85,B 0,C 180,E1 -17844.586,E2 -17844.586} C_VEL
LIN {X 0,Y 270.246,Z 235.82,A -85,B 0,C 180,E1 -17847.911,E2 -17847.911} C_VEL
LIN {X 0,Y 270.159,Z 235.83,A -85,B 0,C 180,E1 -17851.351,E2 -17851.351} C_VEL
LIN {X 0,Y 270.179,Z 235.824,A -85,B 0,C 180,E1 -17854.908,E2 -17854.908} C_VEL
LIN {X 0,Y 270.202,Z 235.813,A -85,B 0,C 180,E1 -17858.72,E2 -17858.72} C_VEL
LIN {X 0,Y 270.193,Z 235.822,A -85,B 0,C 180,E1 -17862.553,E2 -17862.553} C_VEL
LIN {X 0,Y 270.156,Z 235.83,A -85,B 0,C 180,E1 -17866.752,E2 -17866.752} C_VEL
LIN {X 0,Y 270.184,Z 235.827,A -85,B 0,C 180,E1 -17871.293,E2 -17871.293} C_VEL
LIN {X 0,Y 270.19,Z 235.822,A -85,B 0,C 180,E1 -17875.097,E2 -17875.097} C_VEL
LIN {X 0,Y 270.19,Z 235.82,A -85,B 0,C 180,E1 -17879.133,E2 -17879.133} C_VEL
LIN {X 0,Y 270.259,Z 235.819,A -85,B 0,C 180,E1 -17882.147,E2 -17882.147} C_VEL
LIN {X 0,Y 270.27,Z 235.82,A -85,B 0,C 180,E1 -17885.521,E2 -17885.521} C_VEL
LIN {X 0,Y 270.296,Z 235.809,A -85,B 0,C 180,E1 -17890.246,E2 -17890.246} C_VEL
LIN {X 0,Y 270.399,Z 235.801,A -85,B 0,C 180,E1 -17894.937,E2 -17894.937} C_VEL
LIN {X 0,Y 270.439,Z 235.796,A -85,B 0,C 180,E1 -17899.52,E2 -17899.52} C_VEL
LIN {X 0,Y 270.606,Z 235.775,A -85,B 0,C 180,E1 -17902.54,E2 -17902.54} C_VEL
LIN {X 0,Y 270.786,Z 235.752,A -85,B 0,C 180,E1 -17908.513,E2 -17908.513} C_VEL
LIN {X 0,Y 270.785,Z 235.754,A -85,B 0,C 180,E1 -17911.487,E2 -17911.487} C_VEL
LIN {X 0,Y 270.602,Z 235.778,A -85,B 0,C 180,E1 -17917.461,E2 -17917.461} C_VEL
LIN {X 0,Y 270.395,Z 235.803,A -85,B 0,C 180,E1 -17922,E2 -17922} C_VEL
LIN {X 0,Y 270.377,Z 235.804,A -85,B 0,C 180,E1 -17925.899,E2 -17925.899} C_VEL
LIN {X 0,Y 270.286,Z 235.818,A -85,B 0,C 180,E1 -17930.599,E2 -17930.599} C_VEL
LIN {X 0,Y 270.267,Z 235.892,A -85,B 0,C 180,E1 -17932.552,E2 -17932.552} C_VEL
LIN {X 0,Y 272.066,Z 240.69,A -85,B 0,C 180,E1 -17932.857,E2 -17932.857} C_VEL
LIN {X 0,Y 278.437,Z 257.7,A -85,B 0,C 180,E1 -17933.916,E2 -17933.916} C_VEL
LIN {X 0,Y 281.742,Z 268.235,A -85,B 0,C 180,E1 -17934.498,E2 -17934.498} C_VEL
LIN {X 0,Y 279.076,Z 342.712,A -85,B 0,C 180,E1 -17936.699,E2 -17936.699} C_VEL
LIN {X 0,Y 278.273,Z 356.388,A -85,B 0,C 180,E1 -17937.402,E2 -17937.402} C_VEL
LIN {X 0,Y 277.351,Z 369.297,A -85,B 0,C 180,E1 -17938.378,E2 -17938.378} C_VEL
LIN {X 0,Y 276.048,Z 382.231,A -85,B 0,C 180,E1 -17939.696,E2 -17939.696} C_VEL
LIN {X 0,Y 274.738,Z 393.594,A -85,B 0,C 180,E1 -17941.195,E2 -17941.195} C_VEL
LIN {X 0,Y 273.414,Z 403.794,A -85,B 0,C 180,E1 -17942.885,E2 -17942.885} C_VEL
LIN {X 0,Y 272.071,Z 413.408,A -85,B 0,C 180,E1 -17944.852,E2 -17944.852} C_VEL
LIN {X 0,Y 270.792,Z 422.185,A -85,B 0,C 180,E1 -17947.111,E2 -17947.111} C_VEL
LIN {X 0,Y 269.936,Z 428.547,A -85,B 0,C 180,E1 -17949.145,E2 -17949.145} C_VEL
LIN {X 0,Y 269.106,Z 435.013,A -85,B 0,C 180,E1 -17951.758,E2 -17951.758} C_VEL
LIN {X 0,Y 268.634,Z 439.211,A -85,B 0,C 180,E1 -17953.992,E2 -17953.992} C_VEL
LIN {X 0,Y 268.266,Z 442.092,A -85,B 0,C 180,E1 -17956.034,E2 -17956.034} C_VEL
LIN {X 0,Y 268.116,Z 443.382,A -85,B 0,C 180,E1 -17957.212,E2 -17957.212} C_VEL
LIN {X 0,Y 268.033,Z 445.128,A -85,B 0,C 180,E1 -17959.492,E2 -17959.492} C_VEL
LIN {X 0,Y 268.12,Z 445.937,A -85,B 0,C 180,E1 -17961.839,E2 -17961.839} C_VEL
LIN {X 0,Y 268.567,Z 445.537,A -85,B 0,C 180,E1 -17964.852,E2 -17964.852} C_VEL
LIN {X 0,Y 269.051,Z 444.431,A -85,B 0,C 180,E1 -17966.733,E2 -17966.733} C_VEL
LIN {X 0,Y 269.973,Z 441.993,A -85,B 0,C 180,E1 -17969.201,E2 -17969.201} C_VEL
LIN {X 0,Y 271.234,Z 438.19,A -85,B 0,C 180,E1 -17971.749,E2 -17971.749} C_VEL
LIN {X 0,Y 272.881,Z 432.793,A -85,B 0,C 180,E1 -17974.332,E2 -17974.332} C_VEL
LIN {X 0,Y 274.56,Z 427.197,A -85,B 0,C 180,E1 -17976.412,E2 -17976.412} C_VEL
LIN {X 0,Y 276.914,Z 419.047,A -85,B 0,C 180,E1 -17978.798,E2 -17978.798} C_VEL
LIN {X 0,Y 279.207,Z 409.877,A -85,B 0,C 180,E1 -17980.9,E2 -17980.9} C_VEL
LIN {X 0,Y 281.75,Z 399.491,A -85,B 0,C 180,E1 -17982.77,E2 -17982.77} C_VEL
LIN {X 0,Y 284.163,Z 388.185,A -85,B 0,C 180,E1 -17984.356,E2 -17984.356} C_VEL
LIN {X 0,Y 286.104,Z 376.912,A -85,B 0,C 180,E1 -17985.613,E2 -17985.613} C_VEL
LIN {X 0,Y 287.833,Z 365.273,A -85,B 0,C 180,E1 -17986.61,E2 -17986.61} C_VEL
LIN {X 0,Y 289.032,Z 353.219,A -85,B 0,C 180,E1 -17987.39,E2 -17987.39} C_VEL
LIN {X 0,Y 290.076,Z 339.725,A -85,B 0,C 180,E1 -17987.955,E2 -17987.955} C_VEL
LIN {X 0,Y 292.926,Z 286.945,A -85,B 0,C 180,E1 -17989.524,E2 -17989.524} C_VEL
LIN {X 0,Y 292.604,Z 283.876,A -85,B 0,C 180,E1 -17989.694,E2 -17989.694} C_VEL
LIN {X 0,Y 290.945,Z 280.157,A -85,B 0,C 180,E1 -17990.107,E2 -17990.107} C_VEL
LIN {X 0,Y 283.713,Z 271.197,A -85,B 0,C 180,E1 -17991.709,E2 -17991.709} C_VEL
LIN {X 0,Y 277.511,Z 259.325,A -85,B 0,C 180,E1 -17993.411,E2 -17993.411} C_VEL
LIN {X 0,Y 272.326,Z 250.884,A -85,B 0,C 180,E1 -17994.911,E2 -17994.911} C_VEL
LIN {X 0,Y 269.787,Z 247.146,A -85,B 0,C 180,E1 -17995.673,E2 -17995.673} C_VEL
LIN {X 0,Y 264.072,Z 238.432,A -85,B 0,C 180,E1 -17997.617,E2 -17997.617} C_VEL
LIN {X 0,Y 263.702,Z 236.635,A -85,B 0,C 180,E1 -17998.664,E2 -17998.664} C_VEL
LIN {X 0,Y 263.714,Z 236.634,A -85,B 0,C 180,E1 -18001.528,E2 -18001.528} C_VEL
LIN {X 0,Y 263.517,Z 236.659,A -85,B 0,C 180,E1 -18007.664,E2 -18007.664} C_VEL
LIN {X 0,Y 263.321,Z 236.68,A -85,B 0,C 180,E1 -18010.768,E2 -18010.768} C_VEL
LIN {X 0,Y 263.282,Z 236.689,A -85,B 0,C 180,E1 -18015.483,E2 -18015.483} C_VEL
LIN {X 0,Y 263.183,Z 236.695,A -85,B 0,C 180,E1 -18020.314,E2 -18020.314} C_VEL
LIN {X 0,Y 263.164,Z 236.704,A -85,B 0,C 180,E1 -18025.296,E2 -18025.296} C_VEL
LIN {X 0,Y 263.131,Z 236.705,A -85,B 0,C 180,E1 -18028.736,E2 -18028.736} C_VEL
LIN {X 0,Y 263.099,Z 236.706,A -85,B 0,C 180,E1 -18032.294,E2 -18032.294} C_VEL
LIN {X 0,Y 263.141,Z 236.702,A -85,B 0,C 180,E1 -18035.986,E2 -18035.986} C_VEL
LIN {X 0,Y 263.089,Z 236.712,A -85,B 0,C 180,E1 -18039.876,E2 -18039.876} C_VEL
LIN {X 0,Y 263.09,Z 236.711,A -85,B 0,C 180,E1 -18043.992,E2 -18043.992} C_VEL
LIN {X 0,Y 263.113,Z 236.761,A -85,B 0,C 180,E1 -18045.196,E2 -18045.196} C_VEL
LIN {X 0,Y 266.027,Z 245.602,A -85,B 0,C 180,E1 -18050.009,E2 -18050.009} C_VEL
LIN {X 0,Y 268.218,Z 253.132,A -85,B 0,C 180,E1 -18053.508,E2 -18053.508} C_VEL
LIN {X 0,Y 271.18,Z 258.433,A -85,B 0,C 180,E1 -18054.478,E2 -18054.478} C_VEL
LIN {X 0,Y 276.828,Z 269.133,A -85,B 0,C 180,E1 -18056.178,E2 -18056.178} C_VEL
LIN {X 0,Y 282.21,Z 280.846,A -85,B 0,C 180,E1 -18057.713,E2 -18057.713} C_VEL
LIN {X 0,Y 283.277,Z 285.891,A -85,B 0,C 180,E1 -18058.116,E2 -18058.116} C_VEL
LIN {X 0,Y 285.603,Z 302.72,A -85,B 0,C 180,E1 -18059.208,E2 -18059.208} C_VEL
LIN {X 0,Y 286.322,Z 310.733,A -85,B 0,C 180,E1 -18059.641,E2 -18059.641} C_VEL
LIN {X 0,Y 283.234,Z 365.006,A -85,B 0,C 180,E1 -18061.311,E2 -18061.311} C_VEL
LIN {X 0,Y 281.769,Z 379.139,A -85,B 0,C 180,E1 -18062.019,E2 -18062.019} C_VEL
LIN {X 0,Y 279.747,Z 391.812,A -85,B 0,C 180,E1 -18062.916,E2 -18062.916} C_VEL
LIN {X 0,Y 277.419,Z 403.949,A -85,B 0,C 180,E1 -18064.09,E2 -18064.09} C_VEL
LIN {X 0,Y 275.024,Z 414.961,A -85,B 0,C 180,E1 -18065.467,E2 -18065.467} C_VEL
LIN {X 0,Y 272.524,Z 425.064,A -85,B 0,C 180,E1 -18067.045,E2 -18067.045} C_VEL
LIN {X 0,Y 269.795,Z 435.093,A -85,B 0,C 180,E1 -18069.014,E2 -18069.014} C_VEL
LIN {X 0,Y 267.357,Z 444.186,A -85,B 0,C 180,E1 -18071.276,E2 -18071.276} C_VEL
LIN {X 0,Y 265.459,Z 451.151,A -85,B 0,C 180,E1 -18073.467,E2 -18073.467} C_VEL
LIN {X 0,Y 263.453,Z 457.773,A -85,B 0,C 180,E1 -18076.11,E2 -18076.11} C_VEL
LIN {X 0,Y 262.343,Z 462.186,A -85,B 0,C 180,E1 -18078.41,E2 -18078.41} C_VEL
LIN {X 0,Y 261.625,Z 465.547,A -85,B 0,C 180,E1 -18080.726,E2 -18080.726} C_VEL
LIN {X 0,Y 261.316,Z 467.25,A -85,B 0,C 180,E1 -18082.273,E2 -18082.273} C_VEL
LIN {X 0,Y 261.086,Z 469.149,A -85,B 0,C 180,E1 -18084.865,E2 -18084.865} C_VEL
LIN {X 0,Y 261.155,Z 469.808,A -85,B 0,C 180,E1 -18086.915,E2 -18086.915} C_VEL
LIN {X 0,Y 261.196,Z 469.849,A -85,B 0,C 180,E1 -18088.458,E2 -18088.458} C_VEL
LIN {X 0,Y 261.252,Z 469.474,A -85,B 0,C 180,E1 -18090,E2 -18090} C_VEL
LIN {X 0,Y 261.221,Z 468.634,A -85,B 0,C 180,E1 -18091.541,E2 -18091.541} C_VEL
LIN {X 0,Y 261.242,Z 467.379,A -85,B 0,C 180,E1 -18093.084,E2 -18093.084} C_VEL
LIN {X 0,Y 261.264,Z 464.431,A -85,B 0,C 180,E1 -18095.552,E2 -18095.552} C_VEL
LIN {X 0,Y 261.377,Z 460.807,A -85,B 0,C 180,E1 -18097.725,E2 -18097.725} C_VEL
LIN {X 0,Y 261.74,Z 455.777,A -85,B 0,C 180,E1 -18100.05,E2 -18100.05} C_VEL
LIN {X 0,Y 262.394,Z 449.405,A -85,B 0,C 180,E1 -18102.371,E2 -18102.371} C_VEL
LIN {X 0,Y 263.33,Z 442.874,A -85,B 0,C 180,E1 -18104.291,E2 -18104.291} C_VEL
LIN {X 0,Y 264.459,Z 435.008,A -85,B 0,C 180,E1 -18106.201,E2 -18106.201} C_VEL
LIN {X 0,Y 265.465,Z 427.462,A -85,B 0,C 180,E1 -18107.722,E2 -18107.722} C_VEL
LIN {X 0,Y 266.82,Z 417.28,A -85,B 0,C 180,E1 -18109.421,E2 -18109.421} C_VEL
LIN {X 0,Y 268.286,Z 406.017,A -85,B 0,C 180,E1 -18110.909,E2 -18110.909} C_VEL
LIN {X 0,Y 269.884,Z 393.538,A -85,B 0,C 180,E1 -18112.182,E2 -18112.182} C_VEL
LIN {X 0,Y 271.071,Z 380.869,A -85,B 0,C 180,E1 -18113.135,E2 -18113.135} C_VEL
LIN {X 0,Y 272.022,Z 367.963,A -85,B 0,C 180,E1 -18113.806,E2 -18113.806} C_VEL
LIN {X 0,Y 273.67,Z 319.38,A -85,B 0,C 180,E1 -18115.312,E2 -18115.312} C_VEL
LIN {X 0,Y 274.013,Z 306.008,A -85,B 0,C 180,E1 -18115.723,E2 -18115.723} C_VEL
LIN {X 0,Y 268.287,Z 260.554,A -85,B 0,C 180,E1 -18117.674,E2 -18117.674} C_VEL
LIN {X 0,Y 267.591,Z 258.036,A -85,B 0,C 180,E1 -18117.867,E2 -18117.867} C_VEL
LIN {X 0,Y 265.635,Z 248.381,A -85,B 0,C 180,E1 -18121.055,E2 -18121.055} C_VEL
LIN {X 0,Y 263.505,Z 238.273,A -85,B 0,C 180,E1 -18124.533,E2 -18124.533} C_VEL
LIN {X 0,Y 263.179,Z 236.702,A -85,B 0,C 180,E1 -18125.159,E2 -18125.159} C_VEL
LIN {X 0,Y 263.107,Z 236.711,A -85,B 0,C 180,E1 -18129.227,E2 -18129.227} C_VEL
LIN {X 0,Y 263.111,Z 236.713,A -85,B 0,C 180,E1 -18131.89,E2 -18131.89} C_VEL
LIN {X 0,Y 263.09,Z 236.715,A -85,B 0,C 180,E1 -18136.152,E2 -18136.152} C_VEL
LIN {X 0,Y 263.088,Z 236.713,A -85,B 0,C 180,E1 -18140.124,E2 -18140.124} C_VEL
LIN {X 0,Y 263.141,Z 236.706,A -85,B 0,C 180,E1 -18144.014,E2 -18144.014} C_VEL
LIN {X 0,Y 263.098,Z 236.714,A -85,B 0,C 180,E1 -18147.706,E2 -18147.706} C_VEL
LIN {X 0,Y 263.155,Z 236.703,A -85,B 0,C 180,E1 -18151.79,E2 -18151.79} C_VEL
LIN {X 0,Y 263.174,Z 236.7,A -85,B 0,C 180,E1 -18155.211,E2 -18155.211} C_VEL
LIN {X 0,Y 263.181,Z 236.701,A -85,B 0,C 180,E1 -18159.686,E2 -18159.686} C_VEL
LIN {X 0,Y 263.28,Z 236.68,A -85,B 0,C 180,E1 -18164.517,E2 -18164.517} C_VEL
LIN {X 0,Y 263.32,Z 236.686,A -85,B 0,C 180,E1 -18169.232,E2 -18169.232} C_VEL
LIN {X 0,Y 263.518,Z 236.658,A -85,B 0,C 180,E1 -18172.336,E2 -18172.336} C_VEL
LIN {X 0,Y 263.713,Z 236.625,A -85,B 0,C 180,E1 -18178.472,E2 -18178.472} C_VEL
LIN {X 0,Y 263.715,Z 236.627,A -85,B 0,C 180,E1 -18181.527,E2 -18181.527} C_VEL
LIN {X 0,Y 263.521,Z 236.657,A -85,B 0,C 180,E1 -18187.663,E2 -18187.663} C_VEL
LIN {X 0,Y 263.319,Z 236.685,A -85,B 0,C 180,E1 -18190.767,E2 -18190.767} C_VEL
LIN {X 0,Y 263.298,Z 236.676,A -85,B 0,C 180,E1 -18195.481,E2 -18195.481} C_VEL
LIN {X 0,Y 263.262,Z 236.678,A -85,B 0,C 180,E1 -18200.306,E2 -18200.306} C_VEL
LIN {X 0,Y 263.21,Z 236.696,A -85,B 0,C 180,E1 -18204.806,E2 -18204.806} C_VEL
LIN {X 0,Y 263.154,Z 236.705,A -85,B 0,C 180,E1 -18208.732,E2 -18208.732} C_VEL
LIN {X 0,Y 263.108,Z 236.711,A -85,B 0,C 180,E1 -18212.291,E2 -18212.291} C_VEL
LIN {X 0,Y 263.173,Z 236.692,A -85,B 0,C 180,E1 -18216.769,E2 -18216.769} C_VEL
LIN {X 0,Y 263.138,Z 236.692,A -85,B 0,C 180,E1 -18219.866,E2 -18219.866} C_VEL
LIN {X 0,Y 263.121,Z 236.705,A -85,B 0,C 180,E1 -18223.984,E2 -18223.984} C_VEL
LIN {X 0,Y 263.111,Z 236.71,A -85,B 0,C 180,E1 -18228.409,E2 -18228.409} C_VEL
LIN {X 0,Y 263.172,Z 236.699,A -85,B 0,C 180,E1 -18233.239,E2 -18233.239} C_VEL
LIN {X 0,Y 263.122,Z 236.7,A -85,B 0,C 180,E1 -18237.714,E2 -18237.714} C_VEL
LIN {X 0,Y 263.196,Z 236.7,A -85,B 0,C 180,E1 -18241.784,E2 -18241.784} C_VEL
LIN {X 0,Y 263.219,Z 236.697,A -85,B 0,C 180,E1 -18245.203,E2 -18245.203} C_VEL
LIN {X 0,Y 263.258,Z 236.688,A -85,B 0,C 180,E1 -18249.695,E2 -18249.695} C_VEL
LIN {X 0,Y 263.347,Z 236.678,A -85,B 0,C 180,E1 -18254.524,E2 -18254.524} C_VEL
LIN {X 0,Y 263.371,Z 236.678,A -85,B 0,C 180,E1 -18259.236,E2 -18259.236} C_VEL
LIN {X 0,Y 263.568,Z 236.651,A -85,B 0,C 180,E1 -18262.339,E2 -18262.339} C_VEL
LIN {X 0,Y 263.75,Z 236.628,A -85,B 0,C 180,E1 -18268.473,E2 -18268.473} C_VEL
LIN {X 0,Y 263.75,Z 236.63,A -85,B 0,C 180,E1 -18271.527,E2 -18271.527} C_VEL
LIN {X 0,Y 263.56,Z 236.655,A -85,B 0,C 180,E1 -18277.661,E2 -18277.661} C_VEL
LIN {X 0,Y 263.353,Z 236.682,A -85,B 0,C 180,E1 -18280.765,E2 -18280.765} C_VEL
LIN {X 0,Y 263.347,Z 236.681,A -85,B 0,C 180,E1 -18285.477,E2 -18285.477} C_VEL
LIN {X 0,Y 263.257,Z 236.692,A -85,B 0,C 180,E1 -18290.305,E2 -18290.305} C_VEL
LIN {X 0,Y 263.179,Z 236.702,A -85,B 0,C 180,E1 -18291.951,E2 -18291.951} C_VEL
LIN {X 0,Y 265.112,Z 241.766,A -85,B 0,C 180,E1 -18292.32,E2 -18292.32} C_VEL
LIN {X 0,Y 269.936,Z 254.118,A -85,B 0,C 180,E1 -18293.133,E2 -18293.133} C_VEL
LIN {X 0,Y 274.867,Z 268.56,A -85,B 0,C 180,E1 -18293.994,E2 -18293.994} C_VEL
LIN {X 0,Y 272.817,Z 328.648,A -85,B 0,C 180,E1 -18295.795,E2 -18295.795} C_VEL
LIN {X 0,Y 272.092,Z 346.265,A -85,B 0,C 180,E1 -18296.404,E2 -18296.404} C_VEL
LIN {X 0,Y 271.34,Z 359.213,A -85,B 0,C 180,E1 -18297.159,E2 -18297.159} C_VEL
LIN {X 0,Y 270.261,Z 372.391,A -85,B 0,C 180,E1 -18298.248,E2 -18298.248} C_VEL
LIN {X 0,Y 269.021,Z 384.049,A -85,B 0,C 180,E1 -18299.519,E2 -18299.519} C_VEL
LIN {X 0,Y 267.646,Z 395.464,A -85,B 0,C 180,E1 -18301.121,E2 -18301.121} C_VEL
LIN {X 0,Y 266.112,Z 406.438,A -85,B 0,C 180,E1 -18303.05,E2 -18303.05} C_VEL
LIN {X 0,Y 264.724,Z 416.039,A -85,B 0,C 180,E1 -18305.191,E2 -18305.191} C_VEL
LIN {X 0,Y 263.583,Z 423.817,A -85,B 0,C 180,E1 -18307.34,E2 -18307.34} C_VEL
LIN {X 0,Y 262.726,Z 430.144,A -85,B 0,C 180,E1 -18309.503,E2 -18309.503} C_VEL
LIN {X 0,Y 261.915,Z 436.151,A -85,B 0,C 180,E1 -18312.125,E2 -18312.125} C_VEL
LIN {X 0,Y 261.472,Z 440.018,A -85,B 0,C 180,E1 -18314.328,E2 -18314.328} C_VEL
LIN {X 0,Y 261.097,Z 443,A -85,B 0,C 180,E1 -18316.609,E2 -18316.609} C_VEL
LIN {X 0,Y 260.96,Z 445.048,A -85,B 0,C 180,E1 -18318.938,E2 -18318.938} C_VEL
LIN {X 0,Y 261.019,Z 446.229,A -85,B 0,C 180,E1 -18321.737,E2 -18321.737} C_VEL
LIN {X 0,Y 261.289,Z 446.28,A -85,B 0,C 180,E1 -18323.788,E2 -18323.788} C_VEL
LIN {X 0,Y 261.836,Z 445.329,A -85,B 0,C 180,E1 -18326.304,E2 -18326.304} C_VEL
LIN {X 0,Y 262.741,Z 443.217,A -85,B 0,C 180,E1 -18328.856,E2 -18328.856} C_VEL
LIN {X 0,Y 263.975,Z 439.825,A -85,B 0,C 180,E1 -18331.461,E2 -18331.461} C_VEL
LIN {X 0,Y 265.606,Z 434.977,A -85,B 0,C 180,E1 -18334.099,E2 -18334.099} C_VEL
LIN {X 0,Y 267.438,Z 429.436,A -85,B 0,C 180,E1 -18336.376,E2 -18336.376} C_VEL
LIN {X 0,Y 269.57,Z 422.579,A -85,B 0,C 180,E1 -18338.593,E2 -18338.593} C_VEL
LIN {X 0,Y 271.903,Z 414.135,A -85,B 0,C 180,E1 -18340.759,E2 -18340.759} C_VEL
LIN {X 0,Y 274.424,Z 404.707,A -85,B 0,C 180,E1 -18342.68,E2 -18342.68} C_VEL
LIN {X 0,Y 276.684,Z 395.432,A -85,B 0,C 180,E1 -18344.202,E2 -18344.202} C_VEL
LIN {X 0,Y 278.88,Z 384.911,A -85,B 0,C 180,E1 -18345.591,E2 -18345.591} C_VEL
LIN {X 0,Y 281.074,Z 372.139,A -85,B 0,C 180,E1 -18346.904,E2 -18346.904} C_VEL
LIN {X 0,Y 282.597,Z 360.673,A -85,B 0,C 180,E1 -18347.797,E2 -18347.797} C_VEL
LIN {X 0,Y 283.822,Z 348.246,A -85,B 0,C 180,E1 -18348.484,E2 -18348.484} C_VEL
LIN {X 0,Y 284.937,Z 329.507,A -85,B 0,C 180,E1 -18349.13,E2 -18349.13} C_VEL
LIN {X 0,Y 287.81,Z 280.663,A -85,B 0,C 180,E1 -18350.596,E2 -18350.596} C_VEL
LIN {X 0,Y 283.81,Z 271.355,A -85,B 0,C 180,E1 -18351.685,E2 -18351.685} C_VEL
LIN {X 0,Y 283.713,Z 271.197,A -85,B 0,C 180,E1 -18351.709,E2 -18351.709} C_VEL
LIN {X 0,Y 280.782,Z 267.39,A -85,B 0,C 180,E1 -18352.417,E2 -18352.417} C_VEL
LIN {X 0,Y 269.738,Z 257.436,A -85,B 0,C 180,E1 -18355.178,E2 -18355.178} C_VEL
LIN {X 0,Y 267.07,Z 253.74,A -85,B 0,C 180,E1 -18355.994,E2 -18355.994} C_VEL
LIN {X 0,Y 259.583,Z 242.819,A -85,B 0,C 180,E1 -18358.546,E2 -18358.546} C_VEL
LIN {X 0,Y 257.258,Z 239.564,A -85,B 0,C 180,E1 -18359.414,E2 -18359.414} C_VEL
LIN {X 0,Y 256.875,Z 238.404,A -85,B 0,C 180,E1 -18360.001,E2 -18360.001} C_VEL
LIN {X 0,Y 256.69,Z 237.509,A -85,B 0,C 180,E1 -18360.589,E2 -18360.589} C_VEL
LIN {X 0,Y 256.455,Z 237.536,A -85,B 0,C 180,E1 -18363.142,E2 -18363.142} C_VEL
LIN {X 0,Y 256.477,Z 237.534,A -85,B 0,C 180,E1 -18367.875,E2 -18367.875} C_VEL
LIN {X 0,Y 256.229,Z 237.568,A -85,B 0,C 180,E1 -18372.676,E2 -18372.676} C_VEL
LIN {X 0,Y 256.189,Z 237.571,A -85,B 0,C 180,E1 -18376.251,E2 -18376.251} C_VEL
LIN {X 0,Y 256.096,Z 237.58,A -85,B 0,C 180,E1 -18381.1,E2 -18381.1} C_VEL
LIN {X 0,Y 256.145,Z 237.579,A -85,B 0,C 180,E1 -18385.131,E2 -18385.131} C_VEL
LIN {X 0,Y 256.091,Z 237.583,A -85,B 0,C 180,E1 -18388.587,E2 -18388.587} C_VEL
LIN {X 0,Y 256.047,Z 237.588,A -85,B 0,C 180,E1 -18391.701,E2 -18391.701} C_VEL
LIN {X 0,Y 256.062,Z 237.582,A -85,B 0,C 180,E1 -18395.197,E2 -18395.197} C_VEL
LIN {X 0,Y 256.095,Z 237.583,A -85,B 0,C 180,E1 -18397.273,E2 -18397.273} C_VEL
LIN {X 0,Y 256.038,Z 237.588,A -85,B 0,C 180,E1 -18401.207,E2 -18401.207} C_VEL
LIN {X 0,Y 256.032,Z 237.686,A -85,B 0,C 180,E1 -18403.254,E2 -18403.254} C_VEL
LIN {X 0,Y 258.252,Z 244.23,A -85,B 0,C 180,E1 -18407.289,E2 -18407.289} C_VEL
LIN {X 0,Y 260.445,Z 250.994,A -85,B 0,C 180,E1 -18410.878,E2 -18410.878} C_VEL
LIN {X 0,Y 260.99,Z 252.771,A -85,B 0,C 180,E1 -18411.686,E2 -18411.686} C_VEL
LIN {X 0,Y 263.555,Z 257.315,A -85,B 0,C 180,E1 -18412.596,E2 -18412.596} C_VEL
LIN {X 0,Y 264.92,Z 259.473,A -85,B 0,C 180,E1 -18413.053,E2 -18413.053} C_VEL
LIN {X 0,Y 268.229,Z 265.535,A -85,B 0,C 180,E1 -18414.156,E2 -18414.156} C_VEL
LIN {X 0,Y 272.828,Z 274.411,A -85,B 0,C 180,E1 -18415.593,E2 -18415.593} C_VEL
LIN {X 0,Y 277.517,Z 285.069,A -85,B 0,C 180,E1 -18417.021,E2 -18417.021} C_VEL
LIN {X 0,Y 279.875,Z 301.318,A -85,B 0,C 180,E1 -18418.149,E2 -18418.149} C_VEL
LIN {X 0,Y 280.871,Z 310.817,A -85,B 0,C 180,E1 -18418.725,E2 -18418.725} C_VEL
LIN {X 0,Y 277.509,Z 365.605,A -85,B 0,C 180,E1 -18420.462,E2 -18420.462} C_VEL
LIN {X 0,Y 275.997,Z 379.331,A -85,B 0,C 180,E1 -18421.172,E2 -18421.172} C_VEL
LIN {X 0,Y 273.895,Z 391.823,A -85,B 0,C 180,E1 -18422.08,E2 -18422.08} C_VEL
LIN {X 0,Y 271.473,Z 403.89,A -85,B 0,C 180,E1 -18423.272,E2 -18423.272} C_VEL
LIN {X 0,Y 268.957,Z 414.857,A -85,B 0,C 180,E1 -18424.669,E2 -18424.669} C_VEL
LIN {X 0,Y 266.311,Z 424.869,A -85,B 0,C 180,E1 -18426.271,E2 -18426.271} C_VEL
LIN {X 0,Y 263.662,Z 434.007,A -85,B 0,C 180,E1 -18428.091,E2 -18428.091} C_VEL
LIN {X 0,Y 261.106,Z 442.916,A -85,B 0,C 180,E1 -18430.319,E2 -18430.319} C_VEL
LIN {X 0,Y 258.937,Z 450.308,A -85,B 0,C 180,E1 -18432.631,E2 -18432.631} C_VEL
LIN {X 0,Y 257.136,Z 456.195,A -85,B 0,C 180,E1 -18434.952,E2 -18434.952} C_VEL
LIN {X 0,Y 255.661,Z 460.877,A -85,B 0,C 180,E1 -18437.297,E2 -18437.297} C_VEL
LIN {X 0,Y 254.805,Z 464.481,A -85,B 0,C 180,E1 -18439.673,E2 -18439.673} C_VEL
LIN {X 0,Y 254.255,Z 467.089,A -85,B 0,C 180,E1 -18442.057,E2 -18442.057} C_VEL
LIN {X 0,Y 253.985,Z 468.991,A -85,B 0,C 180,E1 -18444.979,E2 -18444.979} C_VEL
LIN {X 0,Y 254.064,Z 469.492,A -85,B 0,C 180,E1 -18446.829,E2 -18446.829} C_VEL
LIN {X 0,Y 254.121,Z 469.492,A -85,B 0,C 180,E1 -18448.415,E2 -18448.415} C_VEL
LIN {X 0,Y 254.174,Z 469.038,A -85,B 0,C 180,E1 -18450,E2 -18450} C_VEL
LIN {X 0,Y 254.147,Z 468.156,A -85,B 0,C 180,E1 -18451.584,E2 -18451.584} C_VEL
LIN {X 0,Y 254.173,Z 466.858,A -85,B 0,C 180,E1 -18453.17,E2 -18453.17} C_VEL
LIN {X 0,Y 254.203,Z 464.032,A -85,B 0,C 180,E1 -18455.551,E2 -18455.551} C_VEL
LIN {X 0,Y 254.322,Z 460.1,A -85,B 0,C 180,E1 -18457.941,E2 -18457.941} C_VEL
LIN {X 0,Y 254.834,Z 453.982,A -85,B 0,C 180,E1 -18460.727,E2 -18460.727} C_VEL
LIN {X 0,Y 255.604,Z 447.205,A -85,B 0,C 180,E1 -18463.109,E2 -18463.109} C_VEL
LIN {X 0,Y 256.784,Z 438.771,A -85,B 0,C 180,E1 -18465.475,E2 -18465.475} C_VEL
LIN {X 0,Y 258.011,Z 430.075,A -85,B 0,C 180,E1 -18467.433,E2 -18467.433} C_VEL
LIN {X 0,Y 259.568,Z 419.35,A -85,B 0,C 180,E1 -18469.368,E2 -18469.368} C_VEL
LIN {X 0,Y 261.069,Z 408.764,A -85,B 0,C 180,E1 -18470.895,E2 -18470.895} C_VEL
LIN {X 0,Y 262.531,Z 397.095,A -85,B 0,C 180,E1 -18472.215,E2 -18472.215} C_VEL
LIN {X 0,Y 263.957,Z 383.932,A -85,B 0,C 180,E1 -18473.329,E2 -18473.329} C_VEL
LIN {X 0,Y 265.01,Z 370.772,A -85,B 0,C 180,E1 -18474.112,E2 -18474.112} C_VEL
LIN {X 0,Y 265.789,Z 354.073,A -85,B 0,C 180,E1 -18474.713,E2 -18474.713} C_VEL
LIN {X 0,Y 267.278,Z 306.667,A -85,B 0,C 180,E1 -18476.193,E2 -18476.193} C_VEL
LIN {X 0,Y 261.819,Z 262.666,A -85,B 0,C 180,E1 -18478.125,E2 -18478.125} C_VEL
LIN {X 0,Y 260.373,Z 257.815,A -85,B 0,C 180,E1 -18478.442,E2 -18478.442} C_VEL
LIN {X 0,Y 257.627,Z 244.381,A -85,B 0,C 180,E1 -18483.061,E2 -18483.061} C_VEL
LIN {X 0,Y 256.126,Z 237.582,A -85,B 0,C 180,E1 -18485.543,E2 -18485.543} C_VEL
LIN {X 0,Y 256.049,Z 237.592,A -85,B 0,C 180,E1 -18489.776,E2 -18489.776} C_VEL
LIN {X 0,Y 256.036,Z 237.593,A -85,B 0,C 180,E1 -18493.326,E2 -18493.326} C_VEL
LIN {X 0,Y 256.054,Z 237.592,A -85,B 0,C 180,E1 -18497.816,E2 -18497.816} C_VEL
LIN {X 0,Y 256.054,Z 237.588,A -85,B 0,C 180,E1 -18500.854,E2 -18500.854} C_VEL
LIN {X 0,Y 256.111,Z 237.581,A -85,B 0,C 180,E1 -18502.863,E2 -18502.863} C_VEL
LIN {X 0,Y 256.043,Z 237.587,A -85,B 0,C 180,E1 -18506.703,E2 -18506.703} C_VEL
LIN {X 0,Y 256.042,Z 237.589,A -85,B 0,C 180,E1 -18510.391,E2 -18510.391} C_VEL
LIN {X 0,Y 256.099,Z 237.579,A -85,B 0,C 180,E1 -18513.954,E2 -18513.954} C_VEL
LIN {X 0,Y 256.049,Z 237.592,A -85,B 0,C 180,E1 -18517.401,E2 -18517.401} C_VEL
LIN {X 0,Y 256.099,Z 237.582,A -85,B 0,C 180,E1 -18520.773,E2 -18520.773} C_VEL
LIN {X 0,Y 256.2,Z 237.56,A -85,B 0,C 180,E1 -18524.078,E2 -18524.078} C_VEL
LIN {X 0,Y 256.261,Z 237.563,A -85,B 0,C 180,E1 -18528.931,E2 -18528.931} C_VEL
LIN {X 0,Y 256.478,Z 237.534,A -85,B 0,C 180,E1 -18532.125,E2 -18532.125} C_VEL
LIN {X 0,Y 256.454,Z 237.533,A -85,B 0,C 180,E1 -18536.858,E2 -18536.858} C_VEL
LIN {X 0,Y 256.709,Z 237.494,A -85,B 0,C 180,E1 -18539.999,E2 -18539.999} C_VEL
LIN {X 0,Y 256.458,Z 237.536,A -85,B 0,C 180,E1 -18543.141,E2 -18543.141} C_VEL
LIN {X 0,Y 256.48,Z 237.534,A -85,B 0,C 180,E1 -18547.874,E2 -18547.874} C_VEL
LIN {X 0,Y 256.229,Z 237.565,A -85,B 0,C 180,E1 -18552.675,E2 -18552.675} C_VEL
LIN {X 0,Y 256.219,Z 237.559,A -85,B 0,C 180,E1 -18556.275,E2 -18556.275} C_VEL
LIN {X 0,Y 256.213,Z 237.559,A -85,B 0,C 180,E1 -18560.891,E2 -18560.891} C_VEL
LIN {X 0,Y 256.17,Z 237.571,A -85,B 0,C 180,E1 -18565.143,E2 -18565.143} C_VEL
LIN {X 0,Y 256.089,Z 237.583,A -85,B 0,C 180,E1 -18569.602,E2 -18569.602} C_VEL
LIN {X 0,Y 256.045,Z 237.586,A -85,B 0,C 180,E1 -18573.295,E2 -18573.295} C_VEL
LIN {X 0,Y 256.103,Z 237.571,A -85,B 0,C 180,E1 -18577.276,E2 -18577.276} C_VEL
LIN {X 0,Y 256.08,Z 237.572,A -85,B 0,C 180,E1 -18581.198,E2 -18581.198} C_VEL
LIN {X 0,Y 256.049,Z 237.586,A -85,B 0,C 180,E1 -18585.531,E2 -18585.531} C_VEL
LIN {X 0,Y 256.041,Z 237.589,A -85,B 0,C 180,E1 -18588.8,E2 -18588.8} C_VEL
LIN {X 0,Y 256.119,Z 237.577,A -85,B 0,C 180,E1 -18592.871,E2 -18592.871} C_VEL
LIN {X 0,Y 256.057,Z 237.577,A -85,B 0,C 180,E1 -18596.71,E2 -18596.71} C_VEL
LIN {X 0,Y 256.107,Z 237.578,A -85,B 0,C 180,E1 -18600.403,E2 -18600.403} C_VEL
LIN {X 0,Y 256.181,Z 237.572,A -85,B 0,C 180,E1 -18604.864,E2 -18604.864} C_VEL
LIN {X 0,Y 256.161,Z 237.573,A -85,B 0,C 180,E1 -18609.107,E2 -18609.107} C_VEL
LIN {X 0,Y 256.296,Z 237.557,A -85,B 0,C 180,E1 -18614.087,E2 -18614.087} C_VEL
LIN {X 0,Y 256.307,Z 237.556,A -85,B 0,C 180,E1 -18618.935,E2 -18618.935} C_VEL
LIN {X 0,Y 256.536,Z 237.527,A -85,B 0,C 180,E1 -18622.128,E2 -18622.128} C_VEL
LIN {X 0,Y 256.713,Z 237.505,A -85,B 0,C 180,E1 -18628.432,E2 -18628.432} C_VEL
LIN {X 0,Y 256.713,Z 237.506,A -85,B 0,C 180,E1 -18631.569,E2 -18631.569} C_VEL
LIN {X 0,Y 256.481,Z 237.534,A -85,B 0,C 180,E1 -18636.292,E2 -18636.292} C_VEL
LIN {X 0,Y 256.424,Z 237.544,A -85,B 0,C 180,E1 -18639.464,E2 -18639.464} C_VEL
LIN {X 0,Y 256.252,Z 237.566,A -85,B 0,C 180,E1 -18644.289,E2 -18644.289} C_VEL
LIN {X 0,Y 256.205,Z 237.57,A -85,B 0,C 180,E1 -18647.56,E2 -18647.56} C_VEL
LIN {X 0,Y 256.181,Z 237.709,A -85,B 0,C 180,E1 -18651.403,E2 -18651.403} C_VEL
LIN {X 0,Y 258.838,Z 244.488,A -85,B 0,C 180,E1 -18651.882,E2 -18651.882} C_VEL
LIN {X 0,Y 263.496,Z 256.367,A -85,B 0,C 180,E1 -18652.694,E2 -18652.694} C_VEL
LIN {X 0,Y 268.21,Z 270.151,A -85,B 0,C 180,E1 -18653.539,E2 -18653.539} C_VEL
LIN {X 0,Y 265.517,Z 343.634,A -85,B 0,C 180,E1 -18655.85,E2 -18655.85} C_VEL
LIN {X 0,Y 264.648,Z 357.308,A -85,B 0,C 180,E1 -18656.594,E2 -18656.594} C_VEL
LIN {X 0,Y 263.669,Z 369.716,A -85,B 0,C 180,E1 -18657.579,E2 -18657.579} C_VEL
LIN {X 0,Y 262.341,Z 382.45,A -85,B 0,C 180,E1 -18658.936,E2 -18658.936} C_VEL
LIN {X 0,Y 260.95,Z 393.716,A -85,B 0,C 180,E1 -18660.478,E2 -18660.478} C_VEL
LIN {X 0,Y 259.498,Z 404.257,A -85,B 0,C 180,E1 -18662.302,E2 -18662.302} C_VEL
LIN {X 0,Y 258.057,Z 414.045,A -85,B 0,C 180,E1 -18664.406,E2 -18664.406} C_VEL
LIN {X 0,Y 256.84,Z 421.998,A -85,B 0,C 180,E1 -18666.529,E2 -18666.529} C_VEL
LIN {X 0,Y 255.716,Z 429.914,A -85,B 0,C 180,E1 -18669.202,E2 -18669.202} C_VEL
LIN {X 0,Y 254.866,Z 436.063,A -85,B 0,C 180,E1 -18671.882,E2 -18671.882} C_VEL
LIN {X 0,Y 254.425,Z 439.953,A -85,B 0,C 180,E1 -18674.095,E2 -18674.095} C_VEL
LIN {X 0,Y 254.052,Z 442.813,A -85,B 0,C 180,E1 -18676.245,E2 -18676.245} C_VEL
LIN {X 0,Y 253.868,Z 444.836,A -85,B 0,C 180,E1 -18678.364,E2 -18678.364} C_VEL
LIN {X 0,Y 253.874,Z 446.243,A -85,B 0,C 180,E1 -18680.809,E2 -18680.809} C_VEL
LIN {X 0,Y 254.107,Z 446.676,A -85,B 0,C 180,E1 -18683.32,E2 -18683.32} C_VEL
LIN {X 0,Y 254.81,Z 445.772,A -85,B 0,C 180,E1 -18686.522,E2 -18686.522} C_VEL
LIN {X 0,Y 255.898,Z 443.409,A -85,B 0,C 180,E1 -18689.464,E2 -18689.464} C_VEL
LIN {X 0,Y 257.366,Z 439.637,A -85,B 0,C 180,E1 -18692.341,E2 -18692.341} C_VEL
LIN {X 0,Y 258.584,Z 436.278,A -85,B 0,C 180,E1 -18694.224,E2 -18694.224} C_VEL
LIN {X 0,Y 260.454,Z 431.02,A -85,B 0,C 180,E1 -18696.541,E2 -18696.541} C_VEL
LIN {X 0,Y 263.081,Z 423.189,A -85,B 0,C 180,E1 -18699.211,E2 -18699.211} C_VEL
LIN {X 0,Y 265.617,Z 414.576,A -85,B 0,C 180,E1 -18701.488,E2 -18701.488} C_VEL
LIN {X 0,Y 268.294,Z 405.238,A -85,B 0,C 180,E1 -18703.433,E2 -18703.433} C_VEL
LIN {X 0,Y 270.943,Z 394.782,A -85,B 0,C 180,E1 -18705.159,E2 -18705.159} C_VEL
LIN {X 0,Y 273.345,Z 383.56,A -85,B 0,C 180,E1 -18706.621,E2 -18706.621} C_VEL
LIN {X 0,Y 275.403,Z 371.837,A -85,B 0,C 180,E1 -18707.818,E2 -18707.818} C_VEL
LIN {X 0,Y 277.23,Z 358.287,A -85,B 0,C 180,E1 -18708.834,E2 -18708.834} C_VEL
LIN {X 0,Y 278.394,Z 345.819,A -85,B 0,C 180,E1 -18709.494,E2 -18709.494} C_VEL
LIN {X 0,Y 282.299,Z 282.598,A -85,B 0,C 180,E1 -18711.488,E2 -18711.488} C_VEL
LIN {X 0,Y 277.13,Z 271.364,A -85,B 0,C 180,E1 -18712.945,E2 -18712.945} C_VEL
LIN {X 0,Y 271.184,Z 260.459,A -85,B 0,C 180,E1 -18714.703,E2 -18714.703} C_VEL
LIN {X 0,Y 267.07,Z 253.74,A -85,B 0,C 180,E1 -18715.994,E2 -18715.994} C_VEL
LIN {X 0,Y 265.333,Z 251.362,A -85,B 0,C 180,E1 -18716.551,E2 -18716.551} C_VEL
LIN {X 0,Y 263.301,Z 249.581,A -85,B 0,C 180,E1 -18717.171,E2 -18717.171} C_VEL
LIN {X 0,Y 258.862,Z 247.133,A -85,B 0,C 180,E1 -18718.523,E2 -18718.523} C_VEL
LIN {X 0,Y 253.456,Z 244.249,A -85,B 0,C 180,E1 -18720.319,E2 -18720.319} C_VEL
LIN {X 0,Y 250.81,Z 241.467,A -85,B 0,C 180,E1 -18721.366,E2 -18721.366} C_VEL
LIN {X 0,Y 249.935,Z 239.891,A -85,B 0,C 180,E1 -18721.813,E2 -18721.813} C_VEL
LIN {X 0,Y 249.425,Z 238.412,A -85,B 0,C 180,E1 -18723.029,E2 -18723.029} C_VEL
LIN {X 0,Y 249.413,Z 238.413,A -85,B 0,C 180,E1 -18726.472,E2 -18726.472} C_VEL
LIN {X 0,Y 249.308,Z 238.43,A -85,B 0,C 180,E1 -18729.738,E2 -18729.738} C_VEL
LIN {X 0,Y 249.142,Z 238.444,A -85,B 0,C 180,E1 -18734.708,E2 -18734.708} C_VEL
LIN {X 0,Y 249.068,Z 238.455,A -85,B 0,C 180,E1 -18738.083,E2 -18738.083} C_VEL
LIN {X 0,Y 249.022,Z 238.464,A -85,B 0,C 180,E1 -18741.525,E2 -18741.525} C_VEL
LIN {X 0,Y 249.091,Z 238.456,A -85,B 0,C 180,E1 -18745.476,E2 -18745.476} C_VEL
LIN {X 0,Y 249.032,Z 238.459,A -85,B 0,C 180,E1 -18748.983,E2 -18748.983} C_VEL
LIN {X 0,Y 248.979,Z 238.464,A -85,B 0,C 180,E1 -18752.434,E2 -18752.434} C_VEL
LIN {X 0,Y 249.011,Z 238.465,A -85,B 0,C 180,E1 -18756.349,E2 -18756.349} C_VEL
LIN {X 0,Y 248.981,Z 238.466,A -85,B 0,C 180,E1 -18760.75,E2 -18760.75} C_VEL
LIN {X 0,Y 250.214,Z 242.056,A -85,B 0,C 180,E1 -18763.497,E2 -18763.497} C_VEL
LIN {X 0,Y 252.345,Z 248.456,A -85,B 0,C 180,E1 -18767.523,E2 -18767.523} C_VEL
LIN {X 0,Y 253.563,Z 252.136,A -85,B 0,C 180,E1 -18769.494,E2 -18769.494} C_VEL
LIN {X 0,Y 256.945,Z 257.464,A -85,B 0,C 180,E1 -18770.82,E2 -18770.82} C_VEL
LIN {X 0,Y 261.449,Z 265.266,A -85,B 0,C 180,E1 -18772.479,E2 -18772.479} C_VEL
LIN {X 0,Y 264.747,Z 271.381,A -85,B 0,C 180,E1 -18773.626,E2 -18773.626} C_VEL
LIN {X 0,Y 270.012,Z 282.084,A -85,B 0,C 180,E1 -18775.35,E2 -18775.35} C_VEL
LIN {X 0,Y 272.725,Z 289.051,A -85,B 0,C 180,E1 -18776.246,E2 -18776.246} C_VEL
LIN {X 0,Y 274.959,Z 306.593,A -85,B 0,C 180,E1 -18777.468,E2 -18777.468} C_VEL
LIN {X 0,Y 275.452,Z 312.441,A -85,B 0,C 180,E1 -18777.814,E2 -18777.814} C_VEL
LIN {X 0,Y 272.086,Z 364.613,A -85,B 0,C 180,E1 -18779.491,E2 -18779.491} C_VEL
LIN {X 0,Y 270.491,Z 378.406,A -85,B 0,C 180,E1 -18780.208,E2 -18780.208} C_VEL
LIN {X 0,Y 268.477,Z 390.03,A -85,B 0,C 180,E1 -18781.038,E2 -18781.038} C_VEL
LIN {X 0,Y 265.919,Z 402.319,A -85,B 0,C 180,E1 -18782.24,E2 -18782.24} C_VEL
LIN {X 0,Y 262.905,Z 414.756,A -85,B 0,C 180,E1 -18783.83,E2 -18783.83} C_VEL
LIN {X 0,Y 259.881,Z 425.686,A -85,B 0,C 180,E1 -18785.647,E2 -18785.647} C_VEL
LIN {X 0,Y 257.127,Z 434.643,A -85,B 0,C 180,E1 -18787.504,E2 -18787.504} C_VEL
LIN {X 0,Y 254.422,Z 443.455,A -85,B 0,C 180,E1 -18789.803,E2 -18789.803} C_VEL
LIN {X 0,Y 252.151,Z 450.546,A -85,B 0,C 180,E1 -18792.148,E2 -18792.148} C_VEL
LIN {X 0,Y 250.262,Z 456.294,A -85,B 0,C 180,E1 -18794.529,E2 -18794.529} C_VEL
LIN {X 0,Y 248.708,Z 460.877,A -85,B 0,C 180,E1 -18796.936,E2 -18796.936} C_VEL
LIN {X 0,Y 247.793,Z 464.39,A -85,B 0,C 180,E1 -18799.378,E2 -18799.378} C_VEL
LIN {X 0,Y 247.194,Z 466.919,A -85,B 0,C 180,E1 -18801.828,E2 -18801.828} C_VEL
LIN {X 0,Y 246.904,Z 468.814,A -85,B 0,C 180,E1 -18805.102,E2 -18805.102} C_VEL
LIN {X 0,Y 246.976,Z 469.176,A -85,B 0,C 180,E1 -18806.738,E2 -18806.738} C_VEL
LIN {X 0,Y 247.047,Z 469.109,A -85,B 0,C 180,E1 -18808.37,E2 -18808.37} C_VEL
LIN {X 0,Y 247.098,Z 468.602,A -85,B 0,C 180,E1 -18810,E2 -18810} C_VEL
LIN {X 0,Y 247.075,Z 467.678,A -85,B 0,C 180,E1 -18811.63,E2 -18811.63} C_VEL
LIN {X 0,Y 247.084,Z 466.335,A -85,B 0,C 180,E1 -18813.261,E2 -18813.261} C_VEL
LIN {X 0,Y 247.131,Z 463.664,A -85,B 0,C 180,E1 -18815.527,E2 -18815.527} C_VEL
LIN {X 0,Y 247.262,Z 459.389,A -85,B 0,C 180,E1 -18818.169,E2 -18818.169} C_VEL
LIN {X 0,Y 247.819,Z 453.112,A -85,B 0,C 180,E1 -18821.035,E2 -18821.035} C_VEL
LIN {X 0,Y 248.669,Z 446.215,A -85,B 0,C 180,E1 -18823.482,E2 -18823.482} C_VEL
LIN {X 0,Y 249.92,Z 437.603,A -85,B 0,C 180,E1 -18825.911,E2 -18825.911} C_VEL
LIN {X 0,Y 251.23,Z 428.7,A -85,B 0,C 180,E1 -18827.92,E2 -18827.92} C_VEL
LIN {X 0,Y 252.641,Z 418.942,A -85,B 0,C 180,E1 -18829.71,E2 -18829.71} C_VEL
LIN {X 0,Y 254.18,Z 408.335,A -85,B 0,C 180,E1 -18831.276,E2 -18831.276} C_VEL
LIN {X 0,Y 255.712,Z 396.637,A -85,B 0,C 180,E1 -18832.627,E2 -18832.627} C_VEL
LIN {X 0,Y 257.155,Z 383.433,A -85,B 0,C 180,E1 -18833.77,E2 -18833.77} C_VEL
LIN {X 0,Y 258.252,Z 370.182,A -85,B 0,C 180,E1 -18834.57,E2 -18834.57} C_VEL
LIN {X 0,Y 259.033,Z 353.371,A -85,B 0,C 180,E1 -18835.187,E2 -18835.187} C_VEL
LIN {X 0,Y 260.526,Z 307.144,A -85,B 0,C 180,E1 -18836.672,E2 -18836.672} C_VEL
LIN {X 0,Y 255.23,Z 264.409,A -85,B 0,C 180,E1 -18838.618,E2 -18838.618} C_VEL
LIN {X 0,Y 253.04,Z 257.511,A -85,B 0,C 180,E1 -18839.086,E2 -18839.086} C_VEL
LIN {X 0,Y 250.577,Z 245.375,A -85,B 0,C 180,E1 -18843.377,E2 -18843.377} C_VEL
LIN {X 0,Y 249.1,Z 238.458,A -85,B 0,C 180,E1 -18846.005,E2 -18846.005} C_VEL
LIN {X 0,Y 248.981,Z 238.47,A -85,B 0,C 180,E1 -18850.477,E2 -18850.477} C_VEL
LIN {X 0,Y 248.988,Z 238.47,A -85,B 0,C 180,E1 -18852.786,E2 -18852.786} C_VEL
LIN {X 0,Y 248.994,Z 238.471,A -85,B 0,C 180,E1 -18857.357,E2 -18857.357} C_VEL
LIN {X 0,Y 249.025,Z 238.464,A -85,B 0,C 180,E1 -18862.197,E2 -18862.197} C_VEL
LIN {X 0,Y 249.023,Z 238.464,A -85,B 0,C 180,E1 -18865.636,E2 -18865.636} C_VEL
LIN {X 0,Y 248.982,Z 238.473,A -85,B 0,C 180,E1 -18869.463,E2 -18869.463} C_VEL
LIN {X 0,Y 249.036,Z 238.461,A -85,B 0,C 180,E1 -18873.157,E2 -18873.157} C_VEL
LIN {X 0,Y 249.03,Z 238.462,A -85,B 0,C 180,E1 -18876.727,E2 -18876.727} C_VEL
LIN {X 0,Y 249.029,Z 238.462,A -85,B 0,C 180,E1 -18880.204,E2 -18880.204} C_VEL
LIN {X 0,Y 249.132,Z 238.442,A -85,B 0,C 180,E1 -18883.614,E2 -18883.614} C_VEL
LIN {X 0,Y 249.204,Z 238.44,A -85,B 0,C 180,E1 -18888.614,E2 -18888.614} C_VEL
LIN {X 0,Y 249.416,Z 238.414,A -85,B 0,C 180,E1 -18891.9,E2 -18891.9} C_VEL
LIN {X 0,Y 249.25,Z 238.432,A -85,B 0,C 180,E1 -18895.147,E2 -18895.147} C_VEL
LIN {X 0,Y 249.638,Z 238.376,A -85,B 0,C 180,E1 -18898.386,E2 -18898.386} C_VEL
LIN {X 0,Y 249.64,Z 238.379,A -85,B 0,C 180,E1 -18901.613,E2 -18901.613} C_VEL
LIN {X 0,Y 249.401,Z 238.415,A -85,B 0,C 180,E1 -18906.823,E2 -18906.823} C_VEL
LIN {X 0,Y 249.306,Z 238.428,A -85,B 0,C 180,E1 -18909.737,E2 -18909.737} C_VEL
LIN {X 0,Y 249.155,Z 238.44,A -85,B 0,C 180,E1 -18914.706,E2 -18914.706} C_VEL
LIN {X 0,Y 249.113,Z 238.436,A -85,B 0,C 180,E1 -18918.079,E2 -18918.079} C_VEL
LIN {X 0,Y 249.116,Z 238.44,A -85,B 0,C 180,E1 -18921.515,E2 -18921.515} C_VEL
LIN {X 0,Y 249.111,Z 238.449,A -85,B 0,C 180,E1 -18925.486,E2 -18925.486} C_VEL
LIN {X 0,Y 249.059,Z 238.459,A -85,B 0,C 180,E1 -18928.995,E2 -18928.995} C_VEL
LIN {X 0,Y 249.008,Z 238.466,A -85,B 0,C 180,E1 -18932.428,E2 -18932.428} C_VEL
LIN {X 0,Y 249.035,Z 238.454,A -85,B 0,C 180,E1 -18936.344,E2 -18936.344} C_VEL
LIN {X 0,Y 249.058,Z 238.446,A -85,B 0,C 180,E1 -18940.467,E2 -18940.467} C_VEL
LIN {X 0,Y 248.996,Z 238.463,A -85,B 0,C 180,E1 -18944.88,E2 -18944.88} C_VEL
LIN {X 0,Y 249.003,Z 238.465,A -85,B 0,C 180,E1 -18947.366,E2 -18947.366} C_VEL
LIN {X 0,Y 249.032,Z 238.462,A -85,B 0,C 180,E1 -18952.203,E2 -18952.203} C_VEL
LIN {X 0,Y 249.033,Z 238.457,A -85,B 0,C 180,E1 -18955.642,E2 -18955.642} C_VEL
LIN {X 0,Y 249.043,Z 238.454,A -85,B 0,C 180,E1 -18959.476,E2 -18959.476} C_VEL
LIN {X 0,Y 249.067,Z 238.458,A -85,B 0,C 180,E1 -18963.165,E2 -18963.165} C_VEL
LIN {X 0,Y 249.073,Z 238.457,A -85,B 0,C 180,E1 -18966.735,E2 -18966.735} C_VEL
LIN {X 0,Y 249.105,Z 238.447,A -85,B 0,C 180,E1 -18970.214,E2 -18970.214} C_VEL
LIN {X 0,Y 249.238,Z 238.438,A -85,B 0,C 180,E1 -18973.624,E2 -18973.624} C_VEL
LIN {X 0,Y 249.25,Z 238.434,A -85,B 0,C 180,E1 -18978.618,E2 -18978.618} C_VEL
LIN {X 0,Y 249.478,Z 238.407,A -85,B 0,C 180,E1 -18981.904,E2 -18981.904} C_VEL
LIN {X 0,Y 249.434,Z 238.413,A -85,B 0,C 180,E1 -18986.77,E2 -18986.77} C_VEL
LIN {X 0,Y 249.727,Z 238.377,A -85,B 0,C 180,E1 -18990,E2 -18990} C_VEL
LIN {X 0,Y 249.434,Z 238.415,A -85,B 0,C 180,E1 -18993.23,E2 -18993.23} C_VEL
LIN {X 0,Y 249.453,Z 238.41,A -85,B 0,C 180,E1 -18996.47,E2 -18996.47} C_VEL
LIN {X 0,Y 249.341,Z 238.426,A -85,B 0,C 180,E1 -18999.736,E2 -18999.736} C_VEL
LIN {X 0,Y 249.202,Z 238.446,A -85,B 0,C 180,E1 -19004.702,E2 -19004.702} C_VEL
LIN {X 0,Y 249.134,Z 238.451,A -85,B 0,C 180,E1 -19008.076,E2 -19008.076} C_VEL
LIN {X 0,Y 249.136,Z 238.453,A -85,B 0,C 180,E1 -19010.79,E2 -19010.79} C_VEL
LIN {X 0,Y 251.716,Z 245.282,A -85,B 0,C 180,E1 -19011.28,E2 -19011.28} C_VEL
LIN {X 0,Y 256.428,Z 256.838,A -85,B 0,C 180,E1 -19012.114,E2 -19012.114} C_VEL
LIN {X 0,Y 261.449,Z 271.412,A -85,B 0,C 180,E1 -19013.047,E2 -19013.047} C_VEL
LIN {X 0,Y 259.351,Z 327.781,A -85,B 0,C 180,E1 -19014.833,E2 -19014.833} C_VEL
LIN {X 0,Y 258.549,Z 346.456,A -85,B 0,C 180,E1 -19015.507,E2 -19015.507} C_VEL
LIN {X 0,Y 257.808,Z 358.411,A -85,B 0,C 180,E1 -19016.214,E2 -19016.214} C_VEL
LIN {X 0,Y 256.729,Z 371.356,A -85,B 0,C 180,E1 -19017.302,E2 -19017.302} C_VEL
LIN {X 0,Y 255.4,Z 383.269,A -85,B 0,C 180,E1 -19018.623,E2 -19018.623} C_VEL
LIN {X 0,Y 254.105,Z 393.51,A -85,B 0,C 180,E1 -19020.061,E2 -19020.061} C_VEL
LIN {X 0,Y 252.616,Z 404.034,A -85,B 0,C 180,E1 -19021.907,E2 -19021.907} C_VEL
LIN {X 0,Y 251.15,Z 413.757,A -85,B 0,C 180,E1 -19024.028,E2 -19024.028} C_VEL
LIN {X 0,Y 249.873,Z 421.813,A -85,B 0,C 180,E1 -19026.199,E2 -19026.199} C_VEL
LIN {X 0,Y 248.72,Z 429.556,A -85,B 0,C 180,E1 -19028.834,E2 -19028.834} C_VEL
LIN {X 0,Y 247.858,Z 435.797,A -85,B 0,C 180,E1 -19031.556,E2 -19031.556} C_VEL
LIN {X 0,Y 247.372,Z 439.797,A -85,B 0,C 180,E1 -19033.821,E2 -19033.821} C_VEL
LIN {X 0,Y 247.108,Z 441.929,A -85,B 0,C 180,E1 -19035.312,E2 -19035.312} C_VEL
LIN {X 0,Y 246.795,Z 444.564,A -85,B 0,C 180,E1 -19037.759,E2 -19037.759} C_VEL
LIN {X 0,Y 246.753,Z 446.261,A -85,B 0,C 180,E1 -19040.258,E2 -19040.258} C_VEL
LIN {X 0,Y 247.04,Z 447.04,A -85,B 0,C 180,E1 -19043.315,E2 -19043.315} C_VEL
